LIN {X -0.244,Y -561.482,Z 954.741,A 0.000,B 0.000,C 90.000,E1 349.398} C_DIS
LIN {X 0.065,Y -565.954,Z 954.738,A 0.000,B 0.000,C 90.000,E1 348.814} C_DIS
LIN {X -0.209,Y -573.077,Z 954.733,A 0.000,B 0.000,C 90.000,E1 347.881} C_DIS
LIN {X -0.280,Y -579.380,Z 954.727,A 0.000,B 0.000,C 90.000,E1 346.937} C_DIS
LIN {X -0.174,Y -584.312,Z 954.723,A 0.000,B 0.000,C 90.000,E1 346.117} C_DIS
LIN {X -0.106,Y -589.678,Z 954.718,A 0.000,B 0.000,C 90.000,E1 345.172} C_DIS
LIN {X 0.183,Y -594.663,Z 954.712,A 0.000,B 0.000,C 90.000,E1 344.212} C_DIS
LIN {X 0.084,Y -600.569,Z 954.706,A 0.000,B 0.000,C 90.000,E1 343.032} C_DIS
LIN {X -0.062,Y -604.887,Z 954.701,A 0.000,B 0.000,C 90.000,E1 342.127} C_DIS
LIN {X 0.073,Y -608.439,Z 954.696,A 0.000,B 0.000,C 90.000,E1 341.329} C_DIS
LIN {X 0.049,Y -611.830,Z 954.692,A 0.000,B 0.000,C 90.000,E1 340.550} C_DIS
LIN {X 0.007,Y -616.058,Z 954.686,A 0.000,B 0.000,C 90.000,E1 339.518} C_DIS
LIN {X 0.265,Y -619.088,Z 954.682,A 0.000,B 0.000,C 90.000,E1 338.720} C_DIS
LIN {X -0.031,Y -622.893,Z 954.676,A 0.000,B 0.000,C 90.000,E1 337.720} C_DIS
LIN {X 0.305,Y -626.443,Z 954.671,A 0.000,B 0.000,C 90.000,E1 336.666} C_DIS
LIN {X 0.111,Y -629.800,Z 954.665,A 0.000,B 0.000,C 90.000,E1 335.665} C_DIS
LIN {X -0.044,Y -632.948,Z 954.659,A 0.000,B 0.000,C 90.000,E1 334.665} C_DIS
LIN {X 0.111,Y -635.819,Z 954.654,A 0.000,B 0.000,C 90.000,E1 333.640} C_DIS
LIN {X -0.205,Y -639.174,Z 954.647,A 0.000,B 0.000,C 90.000,E1 332.410} C_DIS
LIN {X 0.033,Y -641.563,Z 954.641,A 0.000,B 0.000,C 90.000,E1 331.385} C_DIS
LIN {X 0.118,Y -644.440,Z 954.634,A 0.000,B 0.000,C 90.000,E1 330.127} C_DIS
LIN {X 0.253,Y -646.929,Z 954.627,A 0.000,B 0.000,C 90.000,E1 328.869} C_DIS
LIN {X -0.207,Y -648.652,Z 954.622,A 0.000,B 0.000,C 90.000,E1 327.916} C_DIS
LIN {X 0.334,Y -650.629,Z 954.615,A 0.000,B 0.000,C 90.000,E1 326.628} C_DIS
LIN {X 0.361,Y -652.174,Z 954.608,A 0.000,B 0.000,C 90.000,E1 325.388} C_DIS
LIN {X 0.334,Y -653.400,Z 954.602,A 0.000,B 0.000,C 90.000,E1 324.402} C_DIS
LIN {X -0.139,Y -654.470,Z 954.596,A 0.000,B 0.000,C 90.000,E1 323.210} C_DIS
LIN {X 0.253,Y -655.293,Z 954.590,A 0.000,B 0.000,C 90.000,E1 322.190} C_DIS
LIN {X -0.315,Y -656.531,Z 954.581,A 0.000,B 0.000,C 90.000,E1 320.517} C_DIS
LIN {X 0.016,Y -657.478,Z 954.572,A 0.000,B 0.000,C 90.000,E1 319.013} C_DIS
LIN {X 0.167,Y -659.709,Z 954.555,A 0.000,B 0.000,C 90.000,E1 315.810} C_DIS
LIN {X 0.064,Y -660.674,Z 954.548,A 0.000,B 0.000,C 90.000,E1 314.595} C_DIS
LIN {X -0.063,Y -662.179,Z 954.538,A 0.000,B 0.000,C 90.000,E1 312.894} C_DIS
LIN {X 0.363,Y -663.736,Z 954.529,A 0.000,B 0.000,C 90.000,E1 311.148} C_DIS
LIN {X -0.090,Y -664.938,Z 954.521,A 0.000,B 0.000,C 90.000,E1 309.725} C_DIS
LIN {X -0.003,Y -666.013,Z 954.513,A 0.000,B 0.000,C 90.000,E1 308.257} C_DIS
LIN {X 0.022,Y -666.550,Z 954.507,A 0.000,B 0.000,C 90.000,E1 307.282} C_DIS
LIN {X -0.250,Y -667.011,Z 954.500,A 0.000,B 0.000,C 90.000,E1 306.091} C_DIS
LIN {X 0.424,Y -667.346,Z 954.494,A 0.000,B 0.000,C 90.000,E1 304.818} C_DIS
LIN {X -0.038,Y -668.158,Z 954.482,A 0.000,B 0.000,C 90.000,E1 302.673} C_DIS
LIN {X 0.293,Y -669.354,Z 954.469,A 0.000,B 0.000,C 90.000,E1 300.463} C_DIS
LIN {X 0.006,Y -671.420,Z 954.457,A 0.000,B 0.000,C 90.000,E1 298.309} C_DIS
LIN {X -0.153,Y -675.500,Z 954.443,A 0.000,B 0.000,C 90.000,E1 295.668} C_DIS
LIN {X -0.122,Y -677.621,Z 954.436,A 0.000,B 0.000,C 90.000,E1 294.463} C_DIS
LIN {X -0.065,Y -679.550,Z 954.429,A 0.000,B 0.000,C 90.000,E1 293.259} C_DIS
LIN {X 0.055,Y -680.122,Z 954.427,A 0.000,B 0.000,C 90.000,E1 292.770} C_DIS
LIN {X 0.182,Y -680.201,Z 954.424,A 0.000,B 0.000,C 90.000,E1 292.280} C_DIS
LIN {X -0.256,Y -680.187,Z 954.423,A 0.000,B 0.000,C 90.000,E1 292.078} C_DIS
LIN {X -0.319,Y -679.732,Z 954.421,A 0.000,B 0.000,C 90.000,E1 291.844} C_DIS
LIN {X -0.188,Y -678.464,Z 954.419,A 0.000,B 0.000,C 90.000,E1 291.354} C_DIS
LIN {X -0.096,Y -677.859,Z 954.418,A 0.000,B 0.000,C 90.000,E1 291.227} C_DIS
LIN {X 0.086,Y -675.944,Z 954.417,A 0.000,B 0.000,C 90.000,E1 290.972} C_DIS
LIN {X 0.150,Y -672.172,Z 954.415,A 0.000,B 0.000,C 90.000,E1 290.610} C_DIS
LIN {X 0.284,Y -670.597,Z 954.414,A 0.000,B 0.000,C 90.000,E1 290.482} C_DIS
LIN {X 0.022,Y -661.757,Z 954.411,A 0.000,B 0.000,C 90.000,E1 289.939} C_DIS
LIN {X -0.168,Y -659.824,Z 954.410,A 0.000,B 0.000,C 90.000,E1 289.812} C_DIS
LIN {X 0.108,Y -658.940,Z 954.409,A 0.000,B 0.000,C 90.000,E1 289.685} C_DIS
LIN {X 0.072,Y -658.929,Z 954.409,A 0.000,B 0.000,C 90.000,E1 289.685} C_DIS
LIN {X 0.021,Y -658.798,Z 954.409,A 0.000,B 0.000,C 90.000,E1 289.523} C_DIS
LIN {X 0.073,Y -659.029,Z 954.408,A 0.000,B 0.000,C 90.000,E1 289.396} C_DIS
LIN {X 0.012,Y -660.078,Z 954.406,A 0.000,B 0.000,C 90.000,E1 289.033} C_DIS
LIN {X 0.060,Y -663.109,Z 954.402,A 0.000,B 0.000,C 90.000,E1 288.417} C_DIS
LIN {X 0.174,Y -668.460,Z 954.397,A 0.000,B 0.000,C 90.000,E1 287.457} C_DIS
LIN {X 0.095,Y -669.821,Z 954.396,A 0.000,B 0.000,C 90.000,E1 287.221} C_DIS
LIN {X 0.074,Y -673.178,Z 954.392,A 0.000,B 0.000,C 90.000,E1 286.496} C_DIS
LIN {X -0.106,Y -675.937,Z 954.388,A 0.000,B 0.000,C 90.000,E1 285.788} C_DIS
LIN {X -0.029,Y -677.427,Z 954.385,A 0.000,B 0.000,C 90.000,E1 285.300} C_DIS
LIN {X -0.169,Y -679.177,Z 954.381,A 0.000,B 0.000,C 90.000,E1 284.592} C_DIS
LIN {X -0.289,Y -680.537,Z 954.377,A 0.000,B 0.000,C 90.000,E1 283.883} C_DIS
LIN {X 0.233,Y -682.070,Z 954.372,A 0.000,B 0.000,C 90.000,E1 282.883} C_DIS
LIN {X 0.168,Y -682.627,Z 954.369,A 0.000,B 0.000,C 90.000,E1 282.411} C_DIS
LIN {X -0.066,Y -683.123,Z 954.365,A 0.000,B 0.000,C 90.000,E1 281.715} C_DIS
LIN {X -0.125,Y -683.262,Z 954.362,A 0.000,B 0.000,C 90.000,E1 281.243} C_DIS
LIN {X -0.316,Y -683.055,Z 954.360,A 0.000,B 0.000,C 90.000,E1 280.782} C_DIS
LIN {X 0.293,Y -682.648,Z 954.357,A 0.000,B 0.000,C 90.000,E1 280.254} C_DIS
LIN {X 0.106,Y -681.924,Z 954.354,A 0.000,B 0.000,C 90.000,E1 279.792} C_DIS
LIN {X 0.068,Y -681.479,Z 954.353,A 0.000,B 0.000,C 90.000,E1 279.557} C_DIS
LIN {X -0.121,Y -680.255,Z 954.351,A 0.000,B 0.000,C 90.000,E1 279.095} C_DIS
LIN {X -0.213,Y -678.729,Z 954.348,A 0.000,B 0.000,C 90.000,E1 278.624} C_DIS
LIN {X 0.192,Y -675.923,Z 954.344,A 0.000,B 0.000,C 90.000,E1 277.871} C_DIS
LIN {X -0.110,Y -673.075,Z 954.341,A 0.000,B 0.000,C 90.000,E1 277.296} C_DIS
LIN {X 0.317,Y -670.504,Z 954.338,A 0.000,B 0.000,C 90.000,E1 276.777} C_DIS
LIN {X 0.059,Y -667.711,Z 954.335,A 0.000,B 0.000,C 90.000,E1 276.315} C_DIS
LIN {X -0.215,Y -664.623,Z 954.332,A 0.000,B 0.000,C 90.000,E1 275.853} C_DIS
LIN {X 0.058,Y -660.056,Z 954.329,A 0.000,B 0.000,C 90.000,E1 275.220} C_DIS
LIN {X 0.288,Y -654.936,Z 954.326,A 0.000,B 0.000,C 90.000,E1 274.588} C_DIS
LIN {X -0.014,Y -651.703,Z 954.324,A 0.000,B 0.000,C 90.000,E1 274.245} C_DIS
LIN {X 0.194,Y -645.675,Z 954.320,A 0.000,B 0.000,C 90.000,E1 273.612} C_DIS
LIN {X -0.125,Y -639.286,Z 954.317,A 0.000,B 0.000,C 90.000,E1 273.037} C_DIS
LIN {X -0.154,Y -632.639,Z 954.314,A 0.000,B 0.000,C 90.000,E1 272.465} C_DIS
LIN {X -0.117,Y -628.290,Z 954.312,A 0.000,B 0.000,C 90.000,E1 272.121} C_DIS
LIN {X 0.146,Y -623.990,Z 954.310,A 0.000,B 0.000,C 90.000,E1 271.776} C_DIS
LIN {X 0.090,Y -617.979,Z 954.308,A 0.000,B 0.000,C 90.000,E1 271.375} C_DIS
LIN {X -0.084,Y -610.095,Z 954.305,A 0.000,B 0.000,C 90.000,E1 270.917} C_DIS
LIN {X -0.267,Y -603.588,Z 954.303,A 0.000,B 0.000,C 90.000,E1 270.573} C_DIS
LIN {X -0.108,Y -596.754,Z 954.301,A 0.000,B 0.000,C 90.000,E1 270.229} C_DIS
LIN {X -0.054,Y -591.586,Z 954.300,A 0.000,B 0.000,C 90.000,E1 270.000} C_DIS
LIN {X 0.162,Y -584.378,Z 954.299,A 0.000,B 0.000,C 90.000,E1 269.714} C_DIS
LIN {X 0.133,Y -578.913,Z 954.298,A 0.000,B 0.000,C 90.000,E1 269.542} C_DIS
LIN {X -0.182,Y -571.139,Z 954.296,A 0.000,B 0.000,C 90.000,E1 269.370} C_DIS
LIN {X 0.260,Y -564.825,Z 954.296,A 0.000,B 0.000,C 90.000,E1 269.198} C_DIS
LIN {X -0.025,Y -557.881,Z 954.295,A 0.000,B 0.000,C 90.000,E1 269.141} C_DIS
LIN {X 0.065,Y -549.908,Z 954.295,A 0.000,B 0.000,C 90.000,E1 269.083} C_DIS
LIN {X -0.046,Y -548.727,Z 954.295,A 0.000,B 0.000,C 90.000,E1 269.083} C_DIS
LIN {X -0.084,Y -548.413,Z 954.295,A 0.000,B 0.000,C 90.000,E1 269.083} C_DIS
LIN {X -0.218,Y -543.489,Z 954.293,A 0.000,B 0.000,C 90.000,E1 268.740} C_DIS
LIN {X -0.251,Y -543.453,Z 954.293,A 0.000,B 0.000,C 90.000,E1 268.740} C_DIS
LIN {X -0.261,Y -542.935,Z 954.292,A 0.000,B 0.000,C 90.000,E1 268.511} C_DIS
LIN {X -0.023,Y -541.478,Z 954.282,A 0.000,B 0.000,C 90.000,E1 266.731} C_DIS
LIN {X 0.170,Y -540.033,Z 954.271,A 0.000,B 0.000,C 90.000,E1 264.723} C_DIS
LIN {X -0.177,Y -538.999,Z 954.263,A 0.000,B 0.000,C 90.000,E1 263.337} C_DIS
LIN {X -0.003,Y -538.008,Z 954.255,A 0.000,B 0.000,C 90.000,E1 261.894} C_DIS
LIN {X 0.164,Y -536.945,Z 954.249,A 0.000,B 0.000,C 90.000,E1 260.735} C_DIS
LIN {X -0.217,Y -535.611,Z 954.242,A 0.000,B 0.000,C 90.000,E1 259.634} C_DIS
LIN {X 0.199,Y -532.710,Z 954.230,A 0.000,B 0.000,C 90.000,E1 257.297} C_DIS
LIN {X 0.250,Y -529.932,Z 954.217,A 0.000,B 0.000,C 90.000,E1 254.991} C_DIS
LIN {X 0.177,Y -527.986,Z 954.207,A 0.000,B 0.000,C 90.000,E1 253.268} C_DIS
LIN {X 0.204,Y -526.299,Z 954.199,A 0.000,B 0.000,C 90.000,E1 251.819} C_DIS
LIN {X 0.204,Y -524.517,Z 954.191,A 0.000,B 0.000,C 90.000,E1 250.369} C_DIS
LIN {X -0.144,Y -522.628,Z 954.183,A 0.000,B 0.000,C 90.000,E1 248.954} C_DIS
LIN {X 0.112,Y -520.335,Z 954.173,A 0.000,B 0.000,C 90.000,E1 247.177} C_DIS
LIN {X -0.256,Y -518.649,Z 954.167,A 0.000,B 0.000,C 90.000,E1 246.049} C_DIS
LIN {X -0.165,Y -515.883,Z 954.157,A 0.000,B 0.000,C 90.000,E1 244.280} C_DIS
LIN {X -0.022,Y -513.574,Z 954.149,A 0.000,B 0.000,C 90.000,E1 242.794} C_DIS
LIN {X -0.274,Y -510.727,Z 954.139,A 0.000,B 0.000,C 90.000,E1 241.051} C_DIS
LIN {X 0.045,Y -509.196,Z 954.134,A 0.000,B 0.000,C 90.000,E1 240.127} C_DIS
LIN {X 0.187,Y -505.896,Z 954.124,A 0.000,B 0.000,C 90.000,E1 238.329} C_DIS
LIN {X 0.208,Y -502.650,Z 954.116,A 0.000,B 0.000,C 90.000,E1 236.834} C_DIS
LIN {X -0.129,Y -499.952,Z 954.109,A 0.000,B 0.000,C 90.000,E1 235.674} C_DIS
LIN {X -0.085,Y -495.819,Z 954.099,A 0.000,B 0.000,C 90.000,E1 233.863} C_DIS
LIN {X 0.050,Y -493.152,Z 954.093,A 0.000,B 0.000,C 90.000,E1 232.637} C_DIS
LIN {X -0.013,Y -489.753,Z 954.084,A 0.000,B 0.000,C 90.000,E1 231.126} C_DIS
LIN {X -0.212,Y -486.249,Z 954.076,A 0.000,B 0.000,C 90.000,E1 229.622} C_DIS
LIN {X -0.212,Y -481.290,Z 954.064,A 0.000,B 0.000,C 90.000,E1 227.472} C_DIS
LIN {X -0.159,Y -479.200,Z 954.058,A 0.000,B 0.000,C 90.000,E1 226.539} C_DIS
LIN {X -0.249,Y -475.792,Z 954.050,A 0.000,B 0.000,C 90.000,E1 225.000} C_DIS
LIN {X 0.127,Y -470.977,Z 954.038,A 0.000,B 0.000,C 90.000,E1 222.771} C_DIS
LIN {X -0.028,Y -466.887,Z 954.027,A 0.000,B 0.000,C 90.000,E1 220.906} C_DIS
LIN {X 0.167,Y -461.987,Z 954.015,A 0.000,B 0.000,C 90.000,E1 218.669} C_DIS
LIN {X 0.183,Y -458.509,Z 954.006,A 0.000,B 0.000,C 90.000,E1 217.076} C_DIS
LIN {X -0.042,Y -454.181,Z 953.995,A 0.000,B 0.000,C 90.000,E1 215.185} C_DIS
LIN {X 0.015,Y -449.974,Z 953.985,A 0.000,B 0.000,C 90.000,E1 213.245} C_DIS
LIN {X -0.274,Y -445.728,Z 953.974,A 0.000,B 0.000,C 90.000,E1 211.337} C_DIS
LIN {X -0.018,Y -442.885,Z 953.967,A 0.000,B 0.000,C 90.000,E1 210.001} C_DIS
LIN {X -0.117,Y -437.955,Z 953.954,A 0.000,B 0.000,C 90.000,E1 207.719} C_DIS
LIN {X 0.004,Y -434.323,Z 953.945,A 0.000,B 0.000,C 90.000,E1 206.052} C_DIS
LIN {X 0.046,Y -430.643,Z 953.936,A 0.000,B 0.000,C 90.000,E1 204.387} C_DIS
LIN {X 0.017,Y -426.073,Z 953.924,A 0.000,B 0.000,C 90.000,E1 202.386} C_DIS
LIN {X 0.096,Y -419.500,Z 953.908,A 0.000,B 0.000,C 90.000,E1 199.341} C_DIS
LIN {X 0.065,Y -413.978,Z 953.892,A 0.000,B 0.000,C 90.000,E1 196.622} C_DIS
LIN {X 0.135,Y -410.602,Z 953.883,A 0.000,B 0.000,C 90.000,E1 194.898} C_DIS
LIN {X 0.143,Y -406.413,Z 953.871,A 0.000,B 0.000,C 90.000,E1 192.827} C_DIS
LIN {X -0.131,Y -403.062,Z 953.862,A 0.000,B 0.000,C 90.000,E1 191.130} C_DIS
LIN {X -0.067,Y -400.456,Z 953.854,A 0.000,B 0.000,C 90.000,E1 189.726} C_DIS
LIN {X -0.200,Y -397.084,Z 953.844,A 0.000,B 0.000,C 90.000,E1 187.992} C_DIS
LIN {X -0.041,Y -393.117,Z 953.833,A 0.000,B 0.000,C 90.000,E1 185.853} C_DIS
LIN {X -0.021,Y -387.360,Z 953.813,A 0.000,B 0.000,C 90.000,E1 182.293} C_DIS
LIN {X 0.089,Y -386.414,Z 953.807,A 0.000,B 0.000,C 90.000,E1 181.203} C_DIS
LIN {X -0.109,Y -386.020,Z 953.803,A 0.000,B 0.000,C 90.000,E1 180.516} C_DIS
LIN {X 0.177,Y -385.993,Z 953.801,A 0.000,B 0.000,C 90.000,E1 180.115} C_DIS
LIN {X 0.076,Y -386.144,Z 953.799,A 0.000,B 0.000,C 90.000,E1 179.771} C_DIS
LIN {X -0.126,Y -387.039,Z 953.795,A 0.000,B 0.000,C 90.000,E1 179.083} C_DIS
LIN {X 0.071,Y -388.893,Z 953.791,A 0.000,B 0.000,C 90.000,E1 178.339} C_DIS
LIN {X 0.083,Y -390.263,Z 953.789,A 0.000,B 0.000,C 90.000,E1 177.993} C_DIS
LIN {X -0.008,Y -392.230,Z 953.787,A 0.000,B 0.000,C 90.000,E1 177.650} C_DIS
LIN {X -0.092,Y -394.356,Z 953.785,A 0.000,B 0.000,C 90.000,E1 177.306} C_DIS
LIN {X -0.170,Y -397.323,Z 953.783,A 0.000,B 0.000,C 90.000,E1 176.963} C_DIS
LIN {X -0.101,Y -399.882,Z 953.781,A 0.000,B 0.000,C 90.000,E1 176.674} C_DIS
LIN {X -0.205,Y -407.252,Z 953.778,A 0.000,B 0.000,C 90.000,E1 175.988} C_DIS
LIN {X -0.189,Y -413.386,Z 953.775,A 0.000,B 0.000,C 90.000,E1 175.469} C_DIS
LIN {X 0.047,Y -430.440,Z 953.767,A 0.000,B 0.000,C 90.000,E1 173.970} C_DIS
LIN {X -0.025,Y -440.720,Z 953.761,A 0.000,B 0.000,C 90.000,E1 173.053} C_DIS
LIN {X -0.183,Y -449.544,Z 953.757,A 0.000,B 0.000,C 90.000,E1 172.243} C_DIS
LIN {X -0.029,Y -455.300,Z 953.754,A 0.000,B 0.000,C 90.000,E1 171.659} C_DIS
LIN {X -0.017,Y -461.063,Z 953.750,A 0.000,B 0.000,C 90.000,E1 171.084} C_DIS
LIN {X 0.171,Y -470.266,Z 953.745,A 0.000,B 0.000,C 90.000,E1 170.095} C_DIS
LIN {X -0.112,Y -478.133,Z 953.740,A 0.000,B 0.000,C 90.000,E1 169.218} C_DIS
LIN {X 0.139,Y -483.329,Z 953.737,A 0.000,B 0.000,C 90.000,E1 168.578} C_DIS
LIN {X 0.000,Y -489.497,Z 953.732,A 0.000,B 0.000,C 90.000,E1 167.825} C_DIS
LIN {X 0.170,Y -493.049,Z 953.730,A 0.000,B 0.000,C 90.000,E1 167.353} C_DIS
LIN {X -0.085,Y -502.168,Z 953.723,A 0.000,B 0.000,C 90.000,E1 166.172} C_DIS
LIN {X 0.127,Y -509.493,Z 953.717,A 0.000,B 0.000,C 90.000,E1 165.102} C_DIS
LIN {X -0.031,Y -518.221,Z 953.710,A 0.000,B 0.000,C 90.000,E1 163.795} C_DIS
LIN {X -0.104,Y -524.764,Z 953.704,A 0.000,B 0.000,C 90.000,E1 162.779} C_DIS
LIN {X 0.082,Y -532.828,Z 953.697,A 0.000,B 0.000,C 90.000,E1 161.456} C_DIS
LIN {X 0.036,Y -539.926,Z 953.691,A 0.000,B 0.000,C 90.000,E1 160.315} C_DIS
LIN {X 0.218,Y -545.003,Z 953.686,A 0.000,B 0.000,C 90.000,E1 159.444} C_DIS
LIN {X -0.096,Y -552.593,Z 953.679,A 0.000,B 0.000,C 90.000,E1 158.209} C_DIS
LIN {X 0.216,Y -559.724,Z 953.672,A 0.000,B 0.000,C 90.000,E1 156.922} C_DIS
LIN {X 0.218,Y -563.457,Z 953.668,A 0.000,B 0.000,C 90.000,E1 156.230} C_DIS
LIN {X -0.018,Y -569.148,Z 953.662,A 0.000,B 0.000,C 90.000,E1 155.153} C_DIS
LIN {X -0.015,Y -573.176,Z 953.657,A 0.000,B 0.000,C 90.000,E1 154.332} C_DIS
LIN {X -0.270,Y -579.305,Z 953.650,A 0.000,B 0.000,C 90.000,E1 152.999} C_DIS
LIN {X 0.161,Y -582.199,Z 953.646,A 0.000,B 0.000,C 90.000,E1 152.281} C_DIS
LIN {X -0.081,Y -586.471,Z 953.640,A 0.000,B 0.000,C 90.000,E1 151.229} C_DIS
LIN {X 0.251,Y -590.483,Z 953.634,A 0.000,B 0.000,C 90.000,E1 150.127} C_DIS
LIN {X 0.014,Y -595.289,Z 953.627,A 0.000,B 0.000,C 90.000,E1 148.820} C_DIS
LIN {X -0.260,Y -598.936,Z 953.621,A 0.000,B 0.000,C 90.000,E1 147.788} C_DIS
LIN {X -0.061,Y -605.071,Z 953.611,A 0.000,B 0.000,C 90.000,E1 145.928} C_DIS
LIN {X -0.193,Y -608.604,Z 953.605,A 0.000,B 0.000,C 90.000,E1 144.895} C_DIS
LIN {X -0.203,Y -613.893,Z 953.596,A 0.000,B 0.000,C 90.000,E1 143.336} C_DIS
LIN {X -0.289,Y -619.907,Z 953.586,A 0.000,B 0.000,C 90.000,E1 141.537} C_DIS
LIN {X -0.037,Y -624.171,Z 953.579,A 0.000,B 0.000,C 90.000,E1 140.231} C_DIS
LIN {X -0.048,Y -630.122,Z 953.569,A 0.000,B 0.000,C 90.000,E1 138.447} C_DIS
LIN {X 0.103,Y -636.518,Z 953.559,A 0.000,B 0.000,C 90.000,E1 136.662} C_DIS
LIN {X 0.100,Y -641.015,Z 953.552,A 0.000,B 0.000,C 90.000,E1 135.405} C_DIS
LIN {X -0.365,Y -646.462,Z 953.544,A 0.000,B 0.000,C 90.000,E1 133.947} C_DIS
LIN {X -0.264,Y -651.876,Z 953.536,A 0.000,B 0.000,C 90.000,E1 132.447} C_DIS
LIN {X -0.040,Y -658.342,Z 953.526,A 0.000,B 0.000,C 90.000,E1 130.701} C_DIS
LIN {X -0.128,Y -662.979,Z 953.519,A 0.000,B 0.000,C 90.000,E1 129.483} C_DIS
LIN {X -0.047,Y -667.602,Z 953.513,A 0.000,B 0.000,C 90.000,E1 128.257} C_DIS
LIN {X 0.003,Y -671.201,Z 953.507,A 0.000,B 0.000,C 90.000,E1 127.282} C_DIS
LIN {X 0.225,Y -674.629,Z 953.502,A 0.000,B 0.000,C 90.000,E1 126.297} C_DIS
LIN {X -0.054,Y -677.888,Z 953.496,A 0.000,B 0.000,C 90.000,E1 125.358} C_DIS
LIN {X 0.426,Y -681.673,Z 953.490,A 0.000,B 0.000,C 90.000,E1 124.119} C_DIS
LIN {X 0.029,Y -685.100,Z 953.483,A 0.000,B 0.000,C 90.000,E1 122.959} C_DIS
LIN {X 0.054,Y -687.590,Z 953.478,A 0.000,B 0.000,C 90.000,E1 122.005} C_DIS
LIN {X 0.108,Y -689.928,Z 953.473,A 0.000,B 0.000,C 90.000,E1 121.052} C_DIS
LIN {X 0.197,Y -691.468,Z 953.469,A 0.000,B 0.000,C 90.000,E1 120.335} C_DIS
LIN {X 0.069,Y -692.442,Z 953.466,A 0.000,B 0.000,C 90.000,E1 119.873} C_DIS
LIN {X -0.171,Y -694.023,Z 953.461,A 0.000,B 0.000,C 90.000,E1 118.949} C_DIS
LIN {X -0.036,Y -695.058,Z 953.457,A 0.000,B 0.000,C 90.000,E1 118.231} C_DIS
LIN {X 0.363,Y -696.072,Z 953.452,A 0.000,B 0.000,C 90.000,E1 117.257} C_DIS
LIN {X 0.096,Y -696.838,Z 953.445,A 0.000,B 0.000,C 90.000,E1 116.104} C_DIS
LIN {X -0.165,Y -697.205,Z 953.439,A 0.000,B 0.000,C 90.000,E1 114.951} C_DIS
LIN {X 0.321,Y -697.234,Z 953.435,A 0.000,B 0.000,C 90.000,E1 114.207} C_DIS
LIN {X -0.081,Y -696.974,Z 953.432,A 0.000,B 0.000,C 90.000,E1 113.770} C_DIS
LIN {X 0.156,Y -695.919,Z 953.429,A 0.000,B 0.000,C 90.000,E1 113.281} C_DIS
LIN {X -0.230,Y -695.143,Z 953.428,A 0.000,B 0.000,C 90.000,E1 113.078} C_DIS
LIN {X -0.004,Y -692.316,Z 953.426,A 0.000,B 0.000,C 90.000,E1 112.589} C_DIS
LIN {X 0.116,Y -691.505,Z 953.425,A 0.000,B 0.000,C 90.000,E1 112.461} C_DIS
LIN {X 0.235,Y -690.348,Z 953.424,A 0.000,B 0.000,C 90.000,E1 112.333} C_DIS
LIN {X 0.349,Y -688.559,Z 953.424,A 0.000,B 0.000,C 90.000,E1 112.206} C_DIS
LIN {X -0.193,Y -683.327,Z 953.422,A 0.000,B 0.000,C 90.000,E1 111.972} C_DIS
LIN {X -0.287,Y -681.532,Z 953.422,A 0.000,B 0.000,C 90.000,E1 111.897} C_DIS
LIN {X 0.198,Y -677.217,Z 953.421,A 0.000,B 0.000,C 90.000,E1 111.716} C_DIS
LIN {X 0.148,Y -674.161,Z 953.420,A 0.000,B 0.000,C 90.000,E1 111.663} C_DIS
LIN {X 0.387,Y -667.380,Z 953.420,A 0.000,B 0.000,C 90.000,E1 111.589} C_DIS
LIN {X 0.319,Y -632.121,Z 953.420,A 0.000,B 0.000,C 90.000,E1 111.589} C_DIS
LIN {X -0.262,Y -627.805,Z 953.420,A 0.000,B 0.000,C 90.000,E1 111.589} C_DIS
LIN {X 0.027,Y -622.129,Z 953.419,A 0.000,B 0.000,C 90.000,E1 111.461} C_DIS
LIN {X -0.010,Y -615.215,Z 953.418,A 0.000,B 0.000,C 90.000,E1 111.280} C_DIS
LIN {X 0.194,Y -607.245,Z 953.417,A 0.000,B 0.000,C 90.000,E1 110.972} C_DIS
LIN {X -0.121,Y -599.399,Z 953.414,A 0.000,B 0.000,C 90.000,E1 110.610} C_DIS
LIN {X -0.139,Y -594.282,Z 953.413,A 0.000,B 0.000,C 90.000,E1 110.301} C_DIS
LIN {X -0.056,Y -577.074,Z 953.406,A 0.000,B 0.000,C 90.000,E1 109.033} C_DIS
LIN {X 0.286,Y -573.355,Z 953.405,A 0.000,B 0.000,C 90.000,E1 108.779} C_DIS
LIN {X -0.057,Y -568.575,Z 953.403,A 0.000,B 0.000,C 90.000,E1 108.544} C_DIS
LIN {X -0.099,Y -556.788,Z 953.400,A 0.000,B 0.000,C 90.000,E1 108.000} C_DIS
LIN {X -0.205,Y -553.162,Z 953.399,A 0.000,B 0.000,C 90.000,E1 107.819} C_DIS
LIN {X 0.017,Y -551.533,Z 953.398,A 0.000,B 0.000,C 90.000,E1 107.638} C_DIS
LIN {X -0.023,Y -551.496,Z 953.398,A 0.000,B 0.000,C 90.000,E1 107.638} C_DIS
LIN {X 0.100,Y -551.025,Z 953.397,A 0.000,B 0.000,C 90.000,E1 107.402} C_DIS
LIN {X -0.062,Y -550.901,Z 953.394,A 0.000,B 0.000,C 90.000,E1 106.858} C_DIS
LIN {X -0.186,Y -551.549,Z 953.384,A 0.000,B 0.000,C 90.000,E1 105.190} C_DIS
LIN {X 0.043,Y -552.821,Z 953.370,A 0.000,B 0.000,C 90.000,E1 102.647} C_DIS
LIN {X -0.063,Y -554.573,Z 953.358,A 0.000,B 0.000,C 90.000,E1 100.423} C_DIS
LIN {X -0.199,Y -555.592,Z 953.352,A 0.000,B 0.000,C 90.000,E1 99.321} C_DIS
LIN {X -0.135,Y -557.097,Z 953.342,A 0.000,B 0.000,C 90.000,E1 97.644} C_DIS
LIN {X -0.171,Y -558.239,Z 953.335,A 0.000,B 0.000,C 90.000,E1 96.258} C_DIS
LIN {X -0.245,Y -559.174,Z 953.327,A 0.000,B 0.000,C 90.000,E1 94.878} C_DIS
LIN {X -0.214,Y -560.159,Z 953.318,A 0.000,B 0.000,C 90.000,E1 93.212} C_DIS
LIN {X -0.267,Y -560.902,Z 953.310,A 0.000,B 0.000,C 90.000,E1 91.833} C_DIS
LIN {X 0.212,Y -561.512,Z 953.302,A 0.000,B 0.000,C 90.000,E1 90.401} C_DIS
LIN {X 0.045,Y -561.880,Z 953.296,A 0.000,B 0.000,C 90.000,E1 89.312} C_DIS
LIN {X 0.097,Y -562.239,Z 953.287,A 0.000,B 0.000,C 90.000,E1 87.650} C_DIS
LIN {X -0.043,Y -562.489,Z 953.281,A 0.000,B 0.000,C 90.000,E1 86.560} C_DIS
LIN {X -0.042,Y -562.749,Z 953.273,A 0.000,B 0.000,C 90.000,E1 85.179} C_DIS
LIN {X 0.198,Y -563.015,Z 953.263,A 0.000,B 0.000,C 90.000,E1 83.223} C_DIS
LIN {X 0.093,Y -563.492,Z 953.250,A 0.000,B 0.000,C 90.000,E1 81.027} C_DIS
LIN {X -0.210,Y -564.441,Z 953.236,A 0.000,B 0.000,C 90.000,E1 78.578} C_DIS
LIN {X 0.018,Y -565.644,Z 953.224,A 0.000,B 0.000,C 90.000,E1 76.353} C_DIS
LIN {X 0.059,Y -566.723,Z 953.215,A 0.000,B 0.000,C 90.000,E1 74.700} C_DIS
LIN {X 0.054,Y -567.983,Z 953.204,A 0.000,B 0.000,C 90.000,E1 72.779} C_DIS
LIN {X -0.034,Y -568.643,Z 953.198,A 0.000,B 0.000,C 90.000,E1 71.692} C_DIS
LIN {X -0.112,Y -569.260,Z 953.192,A 0.000,B 0.000,C 90.000,E1 70.604} C_DIS
LIN {X 0.158,Y -569.821,Z 953.185,A 0.000,B 0.000,C 90.000,E1 69.209} C_DIS
LIN {X 0.108,Y -570.285,Z 953.177,A 0.000,B 0.000,C 90.000,E1 67.847} C_DIS
LIN {X 0.066,Y -570.668,Z 953.169,A 0.000,B 0.000,C 90.000,E1 66.485} C_DIS
LIN {X 0.087,Y -571.066,Z 953.160,A 0.000,B 0.000,C 90.000,E1 64.845} C_DIS
LIN {X 0.110,Y -571.353,Z 953.151,A 0.000,B 0.000,C 90.000,E1 63.204} C_DIS
LIN {X 0.044,Y -571.509,Z 953.144,A 0.000,B 0.000,C 90.000,E1 61.847} C_DIS
LIN {X 0.086,Y -571.556,Z 953.135,A 0.000,B 0.000,C 90.000,E1 60.205} C_DIS
LIN {X -0.243,Y -571.763,Z 953.124,A 0.000,B 0.000,C 90.000,E1 58.329} C_DIS
LIN {X 0.268,Y -571.663,Z 953.116,A 0.000,B 0.000,C 90.000,E1 56.914} C_DIS
LIN {X -0.182,Y -571.297,Z 953.109,A 0.000,B 0.000,C 90.000,E1 55.595} C_DIS
LIN {X 0.025,Y -570.944,Z 953.103,A 0.000,B 0.000,C 90.000,E1 54.482} C_DIS
LIN {X 0.292,Y -570.754,Z 953.100,A 0.000,B 0.000,C 90.000,E1 53.909} C_DIS
LIN {X -0.107,Y -570.321,Z 953.095,A 0.000,B 0.000,C 90.000,E1 53.130} C_DIS
LIN {X -0.033,Y -569.457,Z 953.089,A 0.000,B 0.000,C 90.000,E1 52.029} C_DIS
LIN {X 0.033,Y -568.445,Z 953.083,A 0.000,B 0.000,C 90.000,E1 50.928} C_DIS
LIN {X 0.082,Y -567.233,Z 953.077,A 0.000,B 0.000,C 90.000,E1 49.828} C_DIS
LIN {X -0.007,Y -566.176,Z 953.072,A 0.000,B 0.000,C 90.000,E1 49.013} C_DIS
LIN {X 0.263,Y -564.866,Z 953.068,A 0.000,B 0.000,C 90.000,E1 48.162} C_DIS
LIN {X 0.199,Y -562.811,Z 953.062,A 0.000,B 0.000,C 90.000,E1 47.067} C_DIS
LIN {X -0.036,Y -561.678,Z 953.059,A 0.000,B 0.000,C 90.000,E1 46.539} C_DIS
LIN {X 0.106,Y -560.484,Z 953.056,A 0.000,B 0.000,C 90.000,E1 45.972} C_DIS
LIN {X -0.090,Y -558.380,Z 953.051,A 0.000,B 0.000,C 90.000,E1 45.162} C_DIS
LIN {X 0.031,Y -556.855,Z 953.048,A 0.000,B 0.000,C 90.000,E1 44.595} C_DIS
LIN {X -0.202,Y -554.269,Z 953.043,A 0.000,B 0.000,C 90.000,E1 43.785} C_DIS
LIN {X -0.114,Y -552.448,Z 953.040,A 0.000,B 0.000,C 90.000,E1 43.218} C_DIS
LIN {X 0.005,Y -549.347,Z 953.035,A 0.000,B 0.000,C 90.000,E1 42.366} C_DIS
LIN {X -0.314,Y -547.132,Z 953.032,A 0.000,B 0.000,C 90.000,E1 41.838} C_DIS
LIN {X 0.320,Y -543.960,Z 953.028,A 0.000,B 0.000,C 90.000,E1 41.067} C_DIS
LIN {X 0.150,Y -540.627,Z 953.024,A 0.000,B 0.000,C 90.000,E1 40.378} C_DIS
LIN {X 0.185,Y -537.684,Z 953.021,A 0.000,B 0.000,C 90.000,E1 39.806} C_DIS
LIN {X -0.211,Y -534.592,Z 953.018,A 0.000,B 0.000,C 90.000,E1 39.277} C_DIS
LIN {X 0.120,Y -531.363,Z 953.015,A 0.000,B 0.000,C 90.000,E1 38.669} C_DIS
LIN {X 0.044,Y -524.446,Z 953.009,A 0.000,B 0.000,C 90.000,E1 37.523} C_DIS
LIN {X 0.104,Y -519.869,Z 953.005,A 0.000,B 0.000,C 90.000,E1 36.790} C_DIS
LIN {X -0.003,Y -516.046,Z 953.001,A 0.000,B 0.000,C 90.000,E1 36.217} C_DIS
LIN {X 0.200,Y -510.042,Z 952.996,A 0.000,B 0.000,C 90.000,E1 35.311} C_DIS
LIN {X -0.081,Y -503.432,Z 952.991,A 0.000,B 0.000,C 90.000,E1 34.452} C_DIS
LIN {X 0.103,Y -498.578,Z 952.988,A 0.000,B 0.000,C 90.000,E1 33.833} C_DIS
LIN {X 0.043,Y -492.112,Z 952.984,A 0.000,B 0.000,C 90.000,E1 33.086} C_DIS
LIN {X 0.146,Y -488.060,Z 952.981,A 0.000,B 0.000,C 90.000,E1 32.625} C_DIS
LIN {X 0.045,Y -481.018,Z 952.977,A 0.000,B 0.000,C 90.000,E1 31.926} C_DIS
LIN {X -0.186,Y -473.908,Z 952.974,A 0.000,B 0.000,C 90.000,E1 31.258} C_DIS
LIN {X 0.243,Y -463.529,Z 952.968,A 0.000,B 0.000,C 90.000,E1 30.256} C_DIS
LIN {X -0.015,Y -456.022,Z 952.965,A 0.000,B 0.000,C 90.000,E1 29.617} C_DIS
LIN {X -0.212,Y -443.997,Z 952.959,A 0.000,B 0.000,C 90.000,E1 28.615} C_DIS
LIN {X 0.107,Y -424.255,Z 952.949,A 0.000,B 0.000,C 90.000,E1 26.873} C_DIS
LIN {X -0.033,Y -407.876,Z 952.941,A 0.000,B 0.000,C 90.000,E1 25.335} C_DIS
LIN {X -0.079,Y -400.514,Z 952.937,A 0.000,B 0.000,C 90.000,E1 24.591} C_DIS
LIN {X -0.012,Y -395.559,Z 952.933,A 0.000,B 0.000,C 90.000,E1 24.003} C_DIS
LIN {X -0.240,Y -393.765,Z 952.932,A 0.000,B 0.000,C 90.000,E1 23.770} C_DIS
LIN {X -0.085,Y -392.059,Z 952.930,A 0.000,B 0.000,C 90.000,E1 23.462} C_DIS
LIN {X 0.014,Y -390.747,Z 952.929,A 0.000,B 0.000,C 90.000,E1 23.131} C_DIS
LIN {X -0.038,Y -390.132,Z 952.927,A 0.000,B 0.000,C 90.000,E1 22.898} C_DIS
LIN {X 0.147,Y -389.392,Z 952.924,A 0.000,B 0.000,C 90.000,E1 22.280} C_DIS
LIN {X 0.037,Y -389.598,Z 952.918,A 0.000,B 0.000,C 90.000,E1 21.227} C_DIS
LIN {X 0.012,Y -394.764,Z 952.888,A 0.000,B 0.000,C 90.000,E1 15.898} C_DIS
LIN {X 0.097,Y -398.370,Z 952.873,A 0.000,B 0.000,C 90.000,E1 13.063} C_DIS
LIN {X 0.125,Y -403.129,Z 952.855,A 0.000,B 0.000,C 90.000,E1 9.905} C_DIS
LIN {X 0.143,Y -406.696,Z 952.844,A 0.000,B 0.000,C 90.000,E1 7.814} C_DIS
LIN {X 0.142,Y -411.909,Z 952.828,A 0.000,B 0.000,C 90.000,E1 5.049} C_DIS
LIN {X -0.164,Y -417.693,Z 952.813,A 0.000,B 0.000,C 90.000,E1 2.350} C_DIS
LIN {X 0.207,Y -424.660,Z 952.797,A 0.000,B 0.000,C 90.000,E1 359.427} C_DIS
LIN {X -0.168,Y -425.684,Z 952.795,A 0.000,B 0.000,C 90.000,E1 359.141} C_DIS
LIN {X -0.105,Y -428.198,Z 952.792,A 0.000,B 0.000,C 90.000,E1 358.568} C_DIS
LIN {X -0.043,Y -430.272,Z 952.790,A 0.000,B 0.000,C 90.000,E1 358.224} C_DIS
LIN {X 0.046,Y -434.368,Z 952.788,A 0.000,B 0.000,C 90.000,E1 357.764} C_DIS
LIN {X 0.051,Y -435.779,Z 952.787,A 0.000,B 0.000,C 90.000,E1 357.650} C_DIS
LIN {X 0.163,Y -440.898,Z 952.785,A 0.000,B 0.000,C 90.000,E1 357.306} C_DIS
LIN {X -0.065,Y -453.945,Z 952.782,A 0.000,B 0.000,C 90.000,E1 356.674} C_DIS
LIN {X -0.028,Y -466.967,Z 952.778,A 0.000,B 0.000,C 90.000,E1 355.988} C_DIS
LIN {X -0.125,Y -480.098,Z 952.774,A 0.000,B 0.000,C 90.000,E1 355.298} C_DIS
LIN {X 0.221,Y -493.049,Z 952.770,A 0.000,B 0.000,C 90.000,E1 354.552} C_DIS
LIN {X 0.224,Y -501.257,Z 952.767,A 0.000,B 0.000,C 90.000,E1 354.090} C_DIS
LIN {X 0.228,Y -510.957,Z 952.764,A 0.000,B 0.000,C 90.000,E1 353.514} C_DIS
LIN {X 0.055,Y -518.522,Z 952.761,A 0.000,B 0.000,C 90.000,E1 353.053} C_DIS
LIN {X 0.234,Y -527.600,Z 952.758,A 0.000,B 0.000,C 90.000,E1 352.413} C_DIS
LIN {X -0.093,Y -536.355,Z 952.754,A 0.000,B 0.000,C 90.000,E1 351.781} C_DIS
LIN {X -0.131,Y -542.080,Z 952.752,A 0.000,B 0.000,C 90.000,E1 351.310} C_DIS
LIN {X -0.274,Y -548.611,Z 952.748,A 0.000,B 0.000,C 90.000,E1 350.735} C_DIS
LIN {X 0.059,Y -555.043,Z 952.745,A 0.000,B 0.000,C 90.000,E1 350.038} C_DIS
LIN {X 0.139,Y -561.125,Z 952.741,A 0.000,B 0.000,C 90.000,E1 349.342} C_DIS
LIN {X -0.107,Y -565.628,Z 952.738,A 0.000,B 0.000,C 90.000,E1 348.814} C_DIS
LIN {X -0.014,Y -570.805,Z 952.734,A 0.000,B 0.000,C 90.000,E1 348.117} C_DIS
LIN {X -0.196,Y -574.694,Z 952.731,A 0.000,B 0.000,C 90.000,E1 347.589} C_DIS
LIN {X -0.007,Y -580.078,Z 952.726,A 0.000,B 0.000,C 90.000,E1 346.756} C_DIS
LIN {X 0.017,Y -585.700,Z 952.721,A 0.000,B 0.000,C 90.000,E1 345.811} C_DIS
LIN {X 0.190,Y -590.326,Z 952.717,A 0.000,B 0.000,C 90.000,E1 344.991} C_DIS
LIN {X -0.010,Y -594.560,Z 952.712,A 0.000,B 0.000,C 90.000,E1 344.212} C_DIS
LIN {X 0.120,Y -599.864,Z 952.706,A 0.000,B 0.000,C 90.000,E1 343.142} C_DIS
LIN {X -0.030,Y -604.256,Z 952.701,A 0.000,B 0.000,C 90.000,E1 342.236} C_DIS
LIN {X -0.087,Y -607.855,Z 952.697,A 0.000,B 0.000,C 90.000,E1 341.456} C_DIS
LIN {X -0.119,Y -611.319,Z 952.693,A 0.000,B 0.000,C 90.000,E1 340.678} C_DIS
LIN {X 0.041,Y -615.558,Z 952.687,A 0.000,B 0.000,C 90.000,E1 339.625} C_DIS
LIN {X 0.076,Y -618.672,Z 952.683,A 0.000,B 0.000,C 90.000,E1 338.847} C_DIS
LIN {X -0.229,Y -622.496,Z 952.677,A 0.000,B 0.000,C 90.000,E1 337.847} C_DIS
LIN {X 0.098,Y -626.140,Z 952.671,A 0.000,B 0.000,C 90.000,E1 336.794} C_DIS
LIN {X -0.102,Y -629.561,Z 952.666,A 0.000,B 0.000,C 90.000,E1 335.793} C_DIS
LIN {X -0.229,Y -633.483,Z 952.658,A 0.000,B 0.000,C 90.000,E1 334.537} C_DIS
LIN {X -0.067,Y -636.347,Z 952.653,A 0.000,B 0.000,C 90.000,E1 333.512} C_DIS
LIN {X 0.193,Y -639.694,Z 952.646,A 0.000,B 0.000,C 90.000,E1 332.231} C_DIS
LIN {X -0.131,Y -642.076,Z 952.640,A 0.000,B 0.000,C 90.000,E1 331.257} C_DIS
LIN {X -0.039,Y -644.945,Z 952.633,A 0.000,B 0.000,C 90.000,E1 329.999} C_DIS
LIN {X 0.026,Y -646.958,Z 952.628,A 0.000,B 0.000,C 90.000,E1 328.997} C_DIS
LIN {X 0.118,Y -648.705,Z 952.622,A 0.000,B 0.000,C 90.000,E1 327.995} C_DIS
LIN {X -0.320,Y -650.331,Z 952.617,A 0.000,B 0.000,C 90.000,E1 327.041} C_DIS
LIN {X -0.276,Y -651.401,Z 952.613,A 0.000,B 0.000,C 90.000,E1 326.294} C_DIS
LIN {X -0.256,Y -653.574,Z 952.603,A 0.000,B 0.000,C 90.000,E1 324.562} C_DIS
LIN {X 0.117,Y -654.489,Z 952.598,A 0.000,B 0.000,C 90.000,E1 323.543} C_DIS
LIN {X 0.116,Y -655.707,Z 952.589,A 0.000,B 0.000,C 90.000,E1 322.065} C_DIS
LIN {X -0.034,Y -656.968,Z 952.580,A 0.000,B 0.000,C 90.000,E1 320.356} C_DIS
LIN {X 0.311,Y -657.904,Z 952.572,A 0.000,B 0.000,C 90.000,E1 318.852} C_DIS
LIN {X -0.424,Y -660.013,Z 952.555,A 0.000,B 0.000,C 90.000,E1 315.972} C_DIS
LIN {X -0.058,Y -660.986,Z 952.548,A 0.000,B 0.000,C 90.000,E1 314.717} C_DIS
LIN {X -0.144,Y -662.248,Z 952.540,A 0.000,B 0.000,C 90.000,E1 313.257} C_DIS
LIN {X 0.274,Y -663.376,Z 952.534,A 0.000,B 0.000,C 90.000,E1 312.000} C_DIS
LIN {X 0.265,Y -664.471,Z 952.527,A 0.000,B 0.000,C 90.000,E1 310.782} C_DIS
LIN {X 0.269,Y -665.467,Z 952.520,A 0.000,B 0.000,C 90.000,E1 309.564} C_DIS
LIN {X 0.361,Y -666.551,Z 952.512,A 0.000,B 0.000,C 90.000,E1 308.096} C_DIS
LIN {X 0.008,Y -666.996,Z 952.508,A 0.000,B 0.000,C 90.000,E1 307.397} C_DIS
LIN {X 0.120,Y -667.546,Z 952.500,A 0.000,B 0.000,C 90.000,E1 305.931} C_DIS
LIN {X -0.134,Y -667.856,Z 952.493,A 0.000,B 0.000,C 90.000,E1 304.739} C_DIS
LIN {X -0.167,Y -668.611,Z 952.482,A 0.000,B 0.000,C 90.000,E1 302.801} C_DIS
LIN {X 0.172,Y -669.793,Z 952.470,A 0.000,B 0.000,C 90.000,E1 300.590} C_DIS
LIN {X 0.063,Y -672.092,Z 952.457,A 0.000,B 0.000,C 90.000,E1 298.180} C_DIS
LIN {X 0.115,Y -676.639,Z 952.441,A 0.000,B 0.000,C 90.000,E1 295.283} C_DIS
LIN {X -0.028,Y -678.295,Z 952.435,A 0.000,B 0.000,C 90.000,E1 294.335} C_DIS
LIN {X -0.155,Y -679.852,Z 952.430,A 0.000,B 0.000,C 90.000,E1 293.387} C_DIS
LIN {X 0.161,Y -680.657,Z 952.426,A 0.000,B 0.000,C 90.000,E1 292.642} C_DIS
LIN {X 0.291,Y -680.615,Z 952.423,A 0.000,B 0.000,C 90.000,E1 292.153} C_DIS
LIN {X -0.147,Y -680.417,Z 952.422,A 0.000,B 0.000,C 90.000,E1 291.950} C_DIS
LIN {X -0.018,Y -679.161,Z 952.419,A 0.000,B 0.000,C 90.000,E1 291.461} C_DIS
LIN {X -0.078,Y -678.100,Z 952.418,A 0.000,B 0.000,C 90.000,E1 291.227} C_DIS
LIN {X 0.014,Y -677.207,Z 952.417,A 0.000,B 0.000,C 90.000,E1 291.099} C_DIS
LIN {X 0.256,Y -672.191,Z 952.415,A 0.000,B 0.000,C 90.000,E1 290.610} C_DIS
LIN {X 0.405,Y -670.668,Z 952.414,A 0.000,B 0.000,C 90.000,E1 290.482} C_DIS
LIN {X 0.041,Y -664.411,Z 952.412,A 0.000,B 0.000,C 90.000,E1 290.120} C_DIS
LIN {X -0.165,Y -660.787,Z 952.410,A 0.000,B 0.000,C 90.000,E1 289.885} C_DIS
LIN {X 0.054,Y -659.322,Z 952.410,A 0.000,B 0.000,C 90.000,E1 289.704} C_DIS
LIN {X 0.020,Y -659.313,Z 952.410,A 0.000,B 0.000,C 90.000,E1 289.704} C_DIS
LIN {X -0.271,Y -659.235,Z 952.409,A 0.000,B 0.000,C 90.000,E1 289.577} C_DIS
LIN {X 0.275,Y -660.197,Z 952.406,A 0.000,B 0.000,C 90.000,E1 289.141} C_DIS
LIN {X 0.110,Y -660.600,Z 952.406,A 0.000,B 0.000,C 90.000,E1 289.033} C_DIS
LIN {X 0.245,Y -663.941,Z 952.402,A 0.000,B 0.000,C 90.000,E1 288.362} C_DIS
LIN {X 0.096,Y -669.368,Z 952.397,A 0.000,B 0.000,C 90.000,E1 287.402} C_DIS
LIN {X 0.020,Y -670.659,Z 952.395,A 0.000,B 0.000,C 90.000,E1 287.166} C_DIS
LIN {X 0.010,Y -673.899,Z 952.391,A 0.000,B 0.000,C 90.000,E1 286.441} C_DIS
LIN {X -0.107,Y -675.770,Z 952.389,A 0.000,B 0.000,C 90.000,E1 285.969} C_DIS
LIN {X -0.079,Y -678.023,Z 952.385,A 0.000,B 0.000,C 90.000,E1 285.245} C_DIS
LIN {X -0.211,Y -679.726,Z 952.381,A 0.000,B 0.000,C 90.000,E1 284.537} C_DIS
LIN {X -0.324,Y -681.078,Z 952.377,A 0.000,B 0.000,C 90.000,E1 283.828} C_DIS
LIN {X 0.240,Y -682.253,Z 952.373,A 0.000,B 0.000,C 90.000,E1 283.063} C_DIS
LIN {X 0.149,Y -683.132,Z 952.369,A 0.000,B 0.000,C 90.000,E1 282.355} C_DIS
LIN {X -0.078,Y -683.629,Z 952.365,A 0.000,B 0.000,C 90.000,E1 281.658} C_DIS
LIN {X -0.134,Y -683.759,Z 952.362,A 0.000,B 0.000,C 90.000,E1 281.186} C_DIS
LIN {X -0.193,Y -683.585,Z 952.359,A 0.000,B 0.000,C 90.000,E1 280.715} C_DIS
LIN {X 0.293,Y -683.161,Z 952.357,A 0.000,B 0.000,C 90.000,E1 280.197} C_DIS
LIN {X 0.225,Y -682.382,Z 952.354,A 0.000,B 0.000,C 90.000,E1 279.726} C_DIS
LIN {X 0.038,Y -681.260,Z 952.352,A 0.000,B 0.000,C 90.000,E1 279.265} C_DIS
LIN {X -0.005,Y -680.643,Z 952.350,A 0.000,B 0.000,C 90.000,E1 279.029} C_DIS
LIN {X -0.200,Y -679.067,Z 952.348,A 0.000,B 0.000,C 90.000,E1 278.568} C_DIS
LIN {X 0.268,Y -677.154,Z 952.345,A 0.000,B 0.000,C 90.000,E1 278.049} C_DIS
LIN {X -0.011,Y -673.847,Z 952.341,A 0.000,B 0.000,C 90.000,E1 277.352} C_DIS
LIN {X -0.328,Y -670.649,Z 952.338,A 0.000,B 0.000,C 90.000,E1 276.777} C_DIS
LIN {X 0.083,Y -667.833,Z 952.335,A 0.000,B 0.000,C 90.000,E1 276.258} C_DIS
LIN {X -0.190,Y -664.711,Z 952.332,A 0.000,B 0.000,C 90.000,E1 275.796} C_DIS
LIN {X 0.175,Y -661.143,Z 952.329,A 0.000,B 0.000,C 90.000,E1 275.277} C_DIS
LIN {X -0.131,Y -657.252,Z 952.327,A 0.000,B 0.000,C 90.000,E1 274.821} C_DIS
LIN {X 0.082,Y -651.803,Z 952.323,A 0.000,B 0.000,C 90.000,E1 274.188} C_DIS
LIN {X 0.251,Y -645.769,Z 952.320,A 0.000,B 0.000,C 90.000,E1 273.555} C_DIS
LIN {X -0.042,Y -640.679,Z 952.317,A 0.000,B 0.000,C 90.000,E1 273.094} C_DIS
LIN {X -0.139,Y -634.030,Z 952.314,A 0.000,B 0.000,C 90.000,E1 272.522} C_DIS
LIN {X -0.082,Y -629.827,Z 952.312,A 0.000,B 0.000,C 90.000,E1 272.178} C_DIS
LIN {X 0.187,Y -623.963,Z 952.310,A 0.000,B 0.000,C 90.000,E1 271.718} C_DIS
LIN {X -0.114,Y -616.588,Z 952.307,A 0.000,B 0.000,C 90.000,E1 271.260} C_DIS
LIN {X 0.219,Y -610.478,Z 952.305,A 0.000,B 0.000,C 90.000,E1 270.859} C_DIS
LIN {X 0.009,Y -603.924,Z 952.303,A 0.000,B 0.000,C 90.000,E1 270.516} C_DIS
LIN {X 0.137,Y -597.098,Z 952.301,A 0.000,B 0.000,C 90.000,E1 270.172} C_DIS
LIN {X 0.154,Y -591.830,Z 952.300,A 0.000,B 0.000,C 90.000,E1 269.943} C_DIS
LIN {X -0.233,Y -584.711,Z 952.298,A 0.000,B 0.000,C 90.000,E1 269.714} C_DIS
LIN {X -0.222,Y -577.303,Z 952.297,A 0.000,B 0.000,C 90.000,E1 269.484} C_DIS
LIN {X 0.044,Y -571.553,Z 952.296,A 0.000,B 0.000,C 90.000,E1 269.312} C_DIS
LIN {X -0.073,Y -565.341,Z 952.296,A 0.000,B 0.000,C 90.000,E1 269.198} C_DIS
LIN {X 0.155,Y -558.224,Z 952.295,A 0.000,B 0.000,C 90.000,E1 269.083} C_DIS
LIN {X 0.117,Y -549.020,Z 952.295,A 0.000,B 0.000,C 90.000,E1 269.026} C_DIS
LIN {X 0.082,Y -548.656,Z 952.295,A 0.000,B 0.000,C 90.000,E1 269.026} C_DIS
LIN {X 0.048,Y -548.351,Z 952.295,A 0.000,B 0.000,C 90.000,E1 269.026} C_DIS
LIN {X 0.086,Y -545.265,Z 952.293,A 0.000,B 0.000,C 90.000,E1 268.797} C_DIS
LIN {X 0.116,Y -543.575,Z 952.293,A 0.000,B 0.000,C 90.000,E1 268.682} C_DIS
LIN {X 0.083,Y -543.532,Z 952.293,A 0.000,B 0.000,C 90.000,E1 268.682} C_DIS
LIN {X -0.111,Y -542.987,Z 952.291,A 0.000,B 0.000,C 90.000,E1 268.453} C_DIS
LIN {X -0.216,Y -541.694,Z 952.283,A 0.000,B 0.000,C 90.000,E1 266.906} C_DIS
LIN {X 0.018,Y -540.194,Z 952.272,A 0.000,B 0.000,C 90.000,E1 264.894} C_DIS
LIN {X 0.152,Y -539.180,Z 952.264,A 0.000,B 0.000,C 90.000,E1 263.457} C_DIS
LIN {X -0.140,Y -538.245,Z 952.256,A 0.000,B 0.000,C 90.000,E1 262.064} C_DIS
LIN {X 0.036,Y -537.214,Z 952.250,A 0.000,B 0.000,C 90.000,E1 260.905} C_DIS
LIN {X 0.132,Y -536.265,Z 952.245,A 0.000,B 0.000,C 90.000,E1 260.038} C_DIS
LIN {X -0.160,Y -534.759,Z 952.238,A 0.000,B 0.000,C 90.000,E1 258.926} C_DIS
LIN {X 0.150,Y -532.622,Z 952.229,A 0.000,B 0.000,C 90.000,E1 257.173} C_DIS
LIN {X 0.209,Y -529.843,Z 952.216,A 0.000,B 0.000,C 90.000,E1 254.866} C_DIS
LIN {X 0.141,Y -527.914,Z 952.206,A 0.000,B 0.000,C 90.000,E1 253.142} C_DIS
LIN {X 0.174,Y -525.866,Z 952.197,A 0.000,B 0.000,C 90.000,E1 251.402} C_DIS
LIN {X 0.173,Y -524.407,Z 952.190,A 0.000,B 0.000,C 90.000,E1 250.242} C_DIS
LIN {X 0.155,Y -522.900,Z 952.184,A 0.000,B 0.000,C 90.000,E1 249.082} C_DIS
LIN {X -0.068,Y -520.628,Z 952.174,A 0.000,B 0.000,C 90.000,E1 247.358} C_DIS
LIN {X 0.046,Y -518.967,Z 952.168,A 0.000,B 0.000,C 90.000,E1 246.177} C_DIS
LIN {X 0.142,Y -516.176,Z 952.158,A 0.000,B 0.000,C 90.000,E1 244.409} C_DIS
LIN {X 0.053,Y -513.862,Z 952.150,A 0.000,B 0.000,C 90.000,E1 242.948} C_DIS
LIN {X 0.042,Y -511.043,Z 952.140,A 0.000,B 0.000,C 90.000,E1 241.179} C_DIS
LIN {X 0.111,Y -509.554,Z 952.135,A 0.000,B 0.000,C 90.000,E1 240.284} C_DIS
LIN {X -0.182,Y -506.274,Z 952.125,A 0.000,B 0.000,C 90.000,E1 238.535} C_DIS
LIN {X -0.153,Y -503.051,Z 952.117,A 0.000,B 0.000,C 90.000,E1 237.041} C_DIS
LIN {X -0.082,Y -501.058,Z 952.112,A 0.000,B 0.000,C 90.000,E1 236.135} C_DIS
LIN {X 0.128,Y -497.613,Z 952.104,A 0.000,B 0.000,C 90.000,E1 234.609} C_DIS
LIN {X -0.280,Y -493.584,Z 952.093,A 0.000,B 0.000,C 90.000,E1 232.844} C_DIS
LIN {X -0.177,Y -489.479,Z 952.083,A 0.000,B 0.000,C 90.000,E1 231.009} C_DIS
LIN {X 0.173,Y -486.726,Z 952.077,A 0.000,B 0.000,C 90.000,E1 229.747} C_DIS
LIN {X -0.133,Y -481.730,Z 952.065,A 0.000,B 0.000,C 90.000,E1 227.634} C_DIS
LIN {X -0.077,Y -479.657,Z 952.059,A 0.000,B 0.000,C 90.000,E1 226.701} C_DIS
LIN {X -0.159,Y -476.262,Z 952.051,A 0.000,B 0.000,C 90.000,E1 225.162} C_DIS
LIN {X 0.317,Y -470.708,Z 952.037,A 0.000,B 0.000,C 90.000,E1 222.609} C_DIS
LIN {X 0.085,Y -467.334,Z 952.028,A 0.000,B 0.000,C 90.000,E1 221.067} C_DIS
LIN {X -0.065,Y -462.430,Z 952.016,A 0.000,B 0.000,C 90.000,E1 218.874} C_DIS
LIN {X -0.064,Y -459.673,Z 952.009,A 0.000,B 0.000,C 90.000,E1 217.604} C_DIS
LIN {X -0.088,Y -456.092,Z 952.000,A 0.000,B 0.000,C 90.000,E1 216.011} C_DIS
LIN {X -0.083,Y -452.498,Z 951.991,A 0.000,B 0.000,C 90.000,E1 214.405} C_DIS
LIN {X 0.226,Y -449.012,Z 951.982,A 0.000,B 0.000,C 90.000,E1 212.752} C_DIS
LIN {X -0.096,Y -444.823,Z 951.971,A 0.000,B 0.000,C 90.000,E1 210.846} C_DIS
LIN {X -0.110,Y -439.104,Z 951.957,A 0.000,B 0.000,C 90.000,E1 208.231} C_DIS
LIN {X 0.206,Y -436.270,Z 951.949,A 0.000,B 0.000,C 90.000,E1 206.873} C_DIS
LIN {X 0.102,Y -431.851,Z 951.938,A 0.000,B 0.000,C 90.000,E1 204.899} C_DIS
LIN {X -0.070,Y -428.864,Z 951.931,A 0.000,B 0.000,C 90.000,E1 203.590} C_DIS
LIN {X -0.122,Y -425.849,Z 951.924,A 0.000,B 0.000,C 90.000,E1 202.259} C_DIS
LIN {X -0.226,Y -419.995,Z 951.909,A 0.000,B 0.000,C 90.000,E1 199.577} C_DIS
LIN {X 0.153,Y -414.439,Z 951.893,A 0.000,B 0.000,C 90.000,E1 196.804} C_DIS
LIN {X -0.034,Y -410.348,Z 951.882,A 0.000,B 0.000,C 90.000,E1 194.773} C_DIS
LIN {X -0.142,Y -406.857,Z 951.872,A 0.000,B 0.000,C 90.000,E1 193.063} C_DIS
LIN {X 0.073,Y -403.492,Z 951.863,A 0.000,B 0.000,C 90.000,E1 191.299} C_DIS
LIN {X 0.060,Y -400.207,Z 951.853,A 0.000,B 0.000,C 90.000,E1 189.557} C_DIS
LIN {X -0.018,Y -396.831,Z 951.843,A 0.000,B 0.000,C 90.000,E1 187.814} C_DIS
LIN {X 0.085,Y -392.877,Z 951.832,A 0.000,B 0.000,C 90.000,E1 185.682} C_DIS
LIN {X 0.098,Y -387.044,Z 951.812,A 0.000,B 0.000,C 90.000,E1 182.121} C_DIS
LIN {X -0.084,Y -386.204,Z 951.808,A 0.000,B 0.000,C 90.000,E1 181.432} C_DIS
LIN {X 0.001,Y -385.558,Z 951.802,A 0.000,B 0.000,C 90.000,E1 180.344} C_DIS
LIN {X 0.182,Y -385.553,Z 951.798,A 0.000,B 0.000,C 90.000,E1 179.599} C_DIS
LIN {X 0.079,Y -385.809,Z 951.796,A 0.000,B 0.000,C 90.000,E1 179.255} C_DIS
LIN {X -0.076,Y -386.602,Z 951.793,A 0.000,B 0.000,C 90.000,E1 178.740} C_DIS
LIN {X 0.159,Y -387.894,Z 951.790,A 0.000,B 0.000,C 90.000,E1 178.167} C_DIS
LIN {X 0.119,Y -389.183,Z 951.788,A 0.000,B 0.000,C 90.000,E1 177.822} C_DIS
LIN {X 0.071,Y -390.016,Z 951.787,A 0.000,B 0.000,C 90.000,E1 177.650} C_DIS
LIN {X -0.106,Y -394.220,Z 951.783,A 0.000,B 0.000,C 90.000,E1 176.963} C_DIS
LIN {X -0.035,Y -400.464,Z 951.779,A 0.000,B 0.000,C 90.000,E1 176.274} C_DIS
LIN {X 0.135,Y -406.308,Z 951.776,A 0.000,B 0.000,C 90.000,E1 175.698} C_DIS
LIN {X 0.152,Y -413.777,Z 951.773,A 0.000,B 0.000,C 90.000,E1 175.065} C_DIS
LIN {X -0.174,Y -427.760,Z 951.766,A 0.000,B 0.000,C 90.000,E1 173.913} C_DIS
LIN {X -0.191,Y -436.865,Z 951.762,A 0.000,B 0.000,C 90.000,E1 173.109} C_DIS
LIN {X -0.015,Y -447.318,Z 951.756,A 0.000,B 0.000,C 90.000,E1 172.129} C_DIS
LIN {X 0.062,Y -457.365,Z 951.751,A 0.000,B 0.000,C 90.000,E1 171.141} C_DIS
LIN {X -0.080,Y -467.325,Z 951.745,A 0.000,B 0.000,C 90.000,E1 170.151} C_DIS
LIN {X -0.038,Y -469.990,Z 951.744,A 0.000,B 0.000,C 90.000,E1 169.859} C_DIS
LIN {X -0.150,Y -479.198,Z 951.738,A 0.000,B 0.000,C 90.000,E1 168.814} C_DIS
LIN {X -0.068,Y -485.493,Z 951.734,A 0.000,B 0.000,C 90.000,E1 168.049} C_DIS
LIN {X -0.135,Y -492.497,Z 951.729,A 0.000,B 0.000,C 90.000,E1 167.173} C_DIS
LIN {X 0.086,Y -501.659,Z 951.722,A 0.000,B 0.000,C 90.000,E1 165.936} C_DIS
LIN {X 0.070,Y -505.876,Z 951.719,A 0.000,B 0.000,C 90.000,E1 165.338} C_DIS
LIN {X 0.242,Y -510.876,Z 951.714,A 0.000,B 0.000,C 90.000,E1 164.574} C_DIS
LIN {X -0.036,Y -515.913,Z 951.710,A 0.000,B 0.000,C 90.000,E1 163.866} C_DIS
LIN {X 0.176,Y -523.464,Z 951.704,A 0.000,B 0.000,C 90.000,E1 162.670} C_DIS
LIN {X -0.167,Y -531.557,Z 951.697,A 0.000,B 0.000,C 90.000,E1 161.402} C_DIS
LIN {X -0.057,Y -538.744,Z 951.690,A 0.000,B 0.000,C 90.000,E1 160.242} C_DIS
LIN {X 0.063,Y -542.970,Z 951.686,A 0.000,B 0.000,C 90.000,E1 159.518} C_DIS
LIN {X 0.218,Y -550.595,Z 951.679,A 0.000,B 0.000,C 90.000,E1 158.230} C_DIS
LIN {X 0.306,Y -557.114,Z 951.673,A 0.000,B 0.000,C 90.000,E1 157.102} C_DIS
LIN {X -0.144,Y -562.448,Z 951.668,A 0.000,B 0.000,C 90.000,E1 156.177} C_DIS
LIN {X 0.020,Y -568.836,Z 951.661,A 0.000,B 0.000,C 90.000,E1 154.921} C_DIS
LIN {X 0.099,Y -572.209,Z 951.657,A 0.000,B 0.000,C 90.000,E1 154.229} C_DIS
LIN {X 0.154,Y -577.792,Z 951.650,A 0.000,B 0.000,C 90.000,E1 152.999} C_DIS
LIN {X -0.282,Y -581.356,Z 951.646,A 0.000,B 0.000,C 90.000,E1 152.231} C_DIS
LIN {X 0.099,Y -584.617,Z 951.641,A 0.000,B 0.000,C 90.000,E1 151.385} C_DIS
LIN {X -0.114,Y -588.762,Z 951.635,A 0.000,B 0.000,C 90.000,E1 150.333} C_DIS
LIN {X -0.079,Y -593.655,Z 951.628,A 0.000,B 0.000,C 90.000,E1 148.997} C_DIS
LIN {X 0.138,Y -597.398,Z 951.622,A 0.000,B 0.000,C 90.000,E1 147.916} C_DIS
LIN {X -0.184,Y -601.824,Z 951.615,A 0.000,B 0.000,C 90.000,E1 146.628} C_DIS
LIN {X -0.102,Y -606.319,Z 951.607,A 0.000,B 0.000,C 90.000,E1 145.308} C_DIS
LIN {X -0.232,Y -612.523,Z 951.597,A 0.000,B 0.000,C 90.000,E1 143.497} C_DIS
LIN {X 0.027,Y -618.611,Z 951.587,A 0.000,B 0.000,C 90.000,E1 141.662} C_DIS
LIN {X 0.266,Y -622.959,Z 951.580,A 0.000,B 0.000,C 90.000,E1 140.356} C_DIS
LIN {X 0.271,Y -632.602,Z 951.564,A 0.000,B 0.000,C 90.000,E1 137.553} C_DIS
LIN {X 0.199,Y -637.194,Z 951.557,A 0.000,B 0.000,C 90.000,E1 136.296} C_DIS
LIN {X -0.257,Y -641.762,Z 951.550,A 0.000,B 0.000,C 90.000,E1 135.081} C_DIS
LIN {X 0.273,Y -646.326,Z 951.543,A 0.000,B 0.000,C 90.000,E1 133.785} C_DIS
LIN {X -0.116,Y -652.727,Z 951.534,A 0.000,B 0.000,C 90.000,E1 132.081} C_DIS
LIN {X 0.135,Y -659.202,Z 951.524,A 0.000,B 0.000,C 90.000,E1 130.334} C_DIS
LIN {X 0.113,Y -665.712,Z 951.515,A 0.000,B 0.000,C 90.000,E1 128.624} C_DIS
LIN {X -0.283,Y -670.323,Z 951.508,A 0.000,B 0.000,C 90.000,E1 127.443} C_DIS
LIN {X -0.071,Y -673.781,Z 951.503,A 0.000,B 0.000,C 90.000,E1 126.457} C_DIS
LIN {X -0.356,Y -677.108,Z 951.497,A 0.000,B 0.000,C 90.000,E1 125.518} C_DIS
LIN {X 0.117,Y -680.941,Z 951.491,A 0.000,B 0.000,C 90.000,E1 124.278} C_DIS
LIN {X 0.088,Y -684.399,Z 951.484,A 0.000,B 0.000,C 90.000,E1 123.086} C_DIS
LIN {X 0.102,Y -686.975,Z 951.479,A 0.000,B 0.000,C 90.000,E1 122.133} C_DIS
LIN {X -0.211,Y -689.298,Z 951.473,A 0.000,B 0.000,C 90.000,E1 121.209} C_DIS
LIN {X 0.227,Y -690.889,Z 951.469,A 0.000,B 0.000,C 90.000,E1 120.463} C_DIS
LIN {X -0.271,Y -692.319,Z 951.465,A 0.000,B 0.000,C 90.000,E1 119.795} C_DIS
LIN {X 0.090,Y -693.838,Z 951.460,A 0.000,B 0.000,C 90.000,E1 118.821} C_DIS
LIN {X 0.224,Y -694.875,Z 951.456,A 0.000,B 0.000,C 90.000,E1 118.103} C_DIS
LIN {X 0.003,Y -695.819,Z 951.451,A 0.000,B 0.000,C 90.000,E1 117.180} C_DIS
LIN {X 0.351,Y -696.513,Z 951.445,A 0.000,B 0.000,C 90.000,E1 115.976} C_DIS
LIN {X 0.084,Y -696.830,Z 951.438,A 0.000,B 0.000,C 90.000,E1 114.823} C_DIS
LIN {X 0.309,Y -696.866,Z 951.435,A 0.000,B 0.000,C 90.000,E1 114.335} C_DIS
LIN {X -0.096,Y -696.657,Z 951.433,A 0.000,B 0.000,C 90.000,E1 113.898} C_DIS
LIN {X 0.161,Y -696.332,Z 951.431,A 0.000,B 0.000,C 90.000,E1 113.643} C_DIS
LIN {X -0.246,Y -695.305,Z 951.429,A 0.000,B 0.000,C 90.000,E1 113.206} C_DIS
LIN {X 0.005,Y -694.179,Z 951.428,A 0.000,B 0.000,C 90.000,E1 112.950} C_DIS
LIN {X 0.104,Y -692.115,Z 951.426,A 0.000,B 0.000,C 90.000,E1 112.589} C_DIS
LIN {X 0.224,Y -691.320,Z 951.425,A 0.000,B 0.000,C 90.000,E1 112.461} C_DIS
LIN {X 0.341,Y -690.170,Z 951.424,A 0.000,B 0.000,C 90.000,E1 112.333} C_DIS
LIN {X -0.179,Y -688.419,Z 951.424,A 0.000,B 0.000,C 90.000,E1 112.259} C_DIS
LIN {X -0.125,Y -681.797,Z 951.422,A 0.000,B 0.000,C 90.000,E1 111.897} C_DIS
LIN {X 0.030,Y -676.791,Z 951.421,A 0.000,B 0.000,C 90.000,E1 111.716} C_DIS
LIN {X 0.141,Y -674.368,Z 951.420,A 0.000,B 0.000,C 90.000,E1 111.663} C_DIS
LIN {X 0.298,Y -667.283,Z 951.420,A 0.000,B 0.000,C 90.000,E1 111.589} C_DIS
LIN {X 0.237,Y -633.015,Z 951.420,A 0.000,B 0.000,C 90.000,E1 111.589} C_DIS
LIN {X -0.285,Y -628.890,Z 951.420,A 0.000,B 0.000,C 90.000,E1 111.589} C_DIS
LIN {X 0.068,Y -623.504,Z 951.419,A 0.000,B 0.000,C 90.000,E1 111.461} C_DIS
LIN {X 0.141,Y -616.533,Z 951.418,A 0.000,B 0.000,C 90.000,E1 111.280} C_DIS
LIN {X 0.031,Y -612.934,Z 951.418,A 0.000,B 0.000,C 90.000,E1 111.173} C_DIS
LIN {X 0.242,Y -607.954,Z 951.417,A 0.000,B 0.000,C 90.000,E1 110.972} C_DIS
LIN {X -0.192,Y -599.704,Z 951.414,A 0.000,B 0.000,C 90.000,E1 110.610} C_DIS
LIN {X 0.171,Y -592.443,Z 951.412,A 0.000,B 0.000,C 90.000,E1 110.120} C_DIS
LIN {X 0.159,Y -576.614,Z 951.405,A 0.000,B 0.000,C 90.000,E1 108.960} C_DIS
LIN {X 0.143,Y -568.152,Z 951.403,A 0.000,B 0.000,C 90.000,E1 108.489} C_DIS
LIN {X 0.256,Y -557.668,Z 951.400,A 0.000,B 0.000,C 90.000,E1 108.000} C_DIS
LIN {X -0.160,Y -553.324,Z 951.399,A 0.000,B 0.000,C 90.000,E1 107.819} C_DIS
LIN {X -0.069,Y -551.566,Z 951.398,A 0.000,B 0.000,C 90.000,E1 107.638} C_DIS
LIN {X -0.102,Y -551.533,Z 951.398,A 0.000,B 0.000,C 90.000,E1 107.638} C_DIS
LIN {X -0.313,Y -551.046,Z 951.397,A 0.000,B 0.000,C 90.000,E1 107.402} C_DIS
LIN {X -0.082,Y -551.089,Z 951.393,A 0.000,B 0.000,C 90.000,E1 106.677} C_DIS
LIN {X 0.220,Y -551.640,Z 951.385,A 0.000,B 0.000,C 90.000,E1 105.245} C_DIS
LIN {X 0.085,Y -552.564,Z 951.374,A 0.000,B 0.000,C 90.000,E1 103.300} C_DIS
LIN {X 0.112,Y -554.362,Z 951.360,A 0.000,B 0.000,C 90.000,E1 100.782} C_DIS
LIN {X 0.203,Y -555.634,Z 951.352,A 0.000,B 0.000,C 90.000,E1 99.378} C_DIS
LIN {X 0.266,Y -557.104,Z 951.343,A 0.000,B 0.000,C 90.000,E1 97.701} C_DIS
LIN {X 0.229,Y -558.233,Z 951.335,A 0.000,B 0.000,C 90.000,E1 96.315} C_DIS
LIN {X -0.053,Y -558.817,Z 951.331,A 0.000,B 0.000,C 90.000,E1 95.511} C_DIS
LIN {X -0.197,Y -559.534,Z 951.324,A 0.000,B 0.000,C 90.000,E1 94.416} C_DIS
LIN {X -0.166,Y -560.482,Z 951.315,A 0.000,B 0.000,C 90.000,E1 92.751} C_DIS
LIN {X -0.241,Y -561.171,Z 951.308,A 0.000,B 0.000,C 90.000,E1 91.375} C_DIS
LIN {X 0.246,Y -561.730,Z 951.300,A 0.000,B 0.000,C 90.000,E1 89.943} C_DIS
LIN {X -0.018,Y -561.966,Z 951.295,A 0.000,B 0.000,C 90.000,E1 89.141} C_DIS
LIN {X 0.034,Y -562.318,Z 951.286,A 0.000,B 0.000,C 90.000,E1 87.478} C_DIS
LIN {X -0.203,Y -562.527,Z 951.281,A 0.000,B 0.000,C 90.000,E1 86.674} C_DIS
LIN {X -0.106,Y -562.806,Z 951.272,A 0.000,B 0.000,C 90.000,E1 85.008} C_DIS
LIN {X 0.129,Y -563.086,Z 951.262,A 0.000,B 0.000,C 90.000,E1 83.053} C_DIS
LIN {X -0.055,Y -563.492,Z 951.251,A 0.000,B 0.000,C 90.000,E1 81.141} C_DIS
LIN {X 0.205,Y -564.448,Z 951.237,A 0.000,B 0.000,C 90.000,E1 78.634} C_DIS
LIN {X -0.111,Y -565.643,Z 951.225,A 0.000,B 0.000,C 90.000,E1 76.464} C_DIS
LIN {X 0.103,Y -566.891,Z 951.214,A 0.000,B 0.000,C 90.000,E1 74.519} C_DIS
LIN {X 0.106,Y -568.138,Z 951.203,A 0.000,B 0.000,C 90.000,E1 72.598} C_DIS
LIN {X -0.018,Y -569.068,Z 951.194,A 0.000,B 0.000,C 90.000,E1 70.967} C_DIS
LIN {X -0.094,Y -569.586,Z 951.188,A 0.000,B 0.000,C 90.000,E1 69.880} C_DIS
LIN {X -0.009,Y -570.185,Z 951.179,A 0.000,B 0.000,C 90.000,E1 68.230} C_DIS
LIN {X -0.233,Y -570.641,Z 951.170,A 0.000,B 0.000,C 90.000,E1 66.613} C_DIS
LIN {X 0.134,Y -571.077,Z 951.159,A 0.000,B 0.000,C 90.000,E1 64.665} C_DIS
LIN {X 0.065,Y -571.303,Z 951.152,A 0.000,B 0.000,C 90.000,E1 63.307} C_DIS
LIN {X -0.259,Y -571.475,Z 951.144,A 0.000,B 0.000,C 90.000,E1 61.975} C_DIS
LIN {X -0.216,Y -571.498,Z 951.135,A 0.000,B 0.000,C 90.000,E1 60.333} C_DIS
LIN {X -0.057,Y -571.704,Z 951.125,A 0.000,B 0.000,C 90.000,E1 58.408} C_DIS
LIN {X -0.031,Y -571.588,Z 951.117,A 0.000,B 0.000,C 90.000,E1 57.041} C_DIS
LIN {X -0.008,Y -571.196,Z 951.109,A 0.000,B 0.000,C 90.000,E1 55.674} C_DIS
LIN {X 0.195,Y -570.844,Z 951.103,A 0.000,B 0.000,C 90.000,E1 54.562} C_DIS
LIN {X -0.204,Y -570.459,Z 951.099,A 0.000,B 0.000,C 90.000,E1 53.783} C_DIS
LIN {X 0.190,Y -569.991,Z 951.094,A 0.000,B 0.000,C 90.000,E1 52.924} C_DIS
LIN {X 0.257,Y -569.100,Z 951.088,A 0.000,B 0.000,C 90.000,E1 51.823} C_DIS
LIN {X 0.314,Y -568.029,Z 951.082,A 0.000,B 0.000,C 90.000,E1 50.723} C_DIS
LIN {X -0.080,Y -566.755,Z 951.076,A 0.000,B 0.000,C 90.000,E1 49.666} C_DIS
LIN {X -0.173,Y -565.633,Z 951.071,A 0.000,B 0.000,C 90.000,E1 48.852} C_DIS
LIN {X -0.009,Y -564.773,Z 951.068,A 0.000,B 0.000,C 90.000,E1 48.286} C_DIS
LIN {X 0.024,Y -562.164,Z 951.061,A 0.000,B 0.000,C 90.000,E1 46.905} C_DIS
LIN {X 0.249,Y -560.362,Z 951.056,A 0.000,B 0.000,C 90.000,E1 46.053} C_DIS
LIN {X 0.052,Y -558.253,Z 951.051,A 0.000,B 0.000,C 90.000,E1 45.243} C_DIS
LIN {X -0.166,Y -555.878,Z 951.047,A 0.000,B 0.000,C 90.000,E1 44.433} C_DIS
LIN {X -0.008,Y -553.216,Z 951.042,A 0.000,B 0.000,C 90.000,E1 43.581} C_DIS
LIN {X 0.075,Y -551.307,Z 951.039,A 0.000,B 0.000,C 90.000,E1 43.014} C_DIS
LIN {X 0.140,Y -549.224,Z 951.036,A 0.000,B 0.000,C 90.000,E1 42.447} C_DIS
LIN {X -0.179,Y -546.986,Z 951.033,A 0.000,B 0.000,C 90.000,E1 41.919} C_DIS
LIN {X -0.313,Y -543.886,Z 951.029,A 0.000,B 0.000,C 90.000,E1 41.229} C_DIS
LIN {X 0.285,Y -540.457,Z 951.025,A 0.000,B 0.000,C 90.000,E1 40.458} C_DIS
LIN {X 0.081,Y -536.745,Z 951.021,A 0.000,B 0.000,C 90.000,E1 39.769} C_DIS
LIN {X -0.079,Y -532.770,Z 951.017,A 0.000,B 0.000,C 90.000,E1 39.072} C_DIS
LIN {X 0.066,Y -528.586,Z 951.013,A 0.000,B 0.000,C 90.000,E1 38.338} C_DIS
LIN {X 0.137,Y -522.424,Z 951.007,A 0.000,B 0.000,C 90.000,E1 37.317} C_DIS
LIN {X 0.178,Y -517.744,Z 951.003,A 0.000,B 0.000,C 90.000,E1 36.583} C_DIS
LIN {X -0.016,Y -511.775,Z 950.999,A 0.000,B 0.000,C 90.000,E1 35.724} C_DIS
LIN {X 0.234,Y -507.552,Z 950.995,A 0.000,B 0.000,C 90.000,E1 35.105} C_DIS
LIN {X -0.158,Y -501.920,Z 950.991,A 0.000,B 0.000,C 90.000,E1 34.405} C_DIS
LIN {X 0.018,Y -496.996,Z 950.988,A 0.000,B 0.000,C 90.000,E1 33.785} C_DIS
LIN {X 0.041,Y -490.414,Z 950.984,A 0.000,B 0.000,C 90.000,E1 33.038} C_DIS
LIN {X -0.239,Y -486.249,Z 950.981,A 0.000,B 0.000,C 90.000,E1 32.625} C_DIS
LIN {X 0.105,Y -479.220,Z 950.977,A 0.000,B 0.000,C 90.000,E1 31.878} C_DIS
LIN {X -0.035,Y -473.456,Z 950.974,A 0.000,B 0.000,C 90.000,E1 31.337} C_DIS
LIN {X -0.014,Y -463.061,Z 950.969,A 0.000,B 0.000,C 90.000,E1 30.384} C_DIS
LIN {X -0.014,Y -455.532,Z 950.965,A 0.000,B 0.000,C 90.000,E1 29.716} C_DIS
LIN {X -0.147,Y -444.849,Z 950.960,A 0.000,B 0.000,C 90.000,E1 28.821} C_DIS
LIN {X 0.123,Y -424.991,Z 950.951,A 0.000,B 0.000,C 90.000,E1 27.078} C_DIS
LIN {X -0.014,Y -410.316,Z 950.943,A 0.000,B 0.000,C 90.000,E1 25.720} C_DIS
LIN {X -0.118,Y -400.108,Z 950.937,A 0.000,B 0.000,C 90.000,E1 24.695} C_DIS
LIN {X 0.184,Y -397.292,Z 950.935,A 0.000,B 0.000,C 90.000,E1 24.335} C_DIS
LIN {X 0.124,Y -393.895,Z 950.933,A 0.000,B 0.000,C 90.000,E1 23.898} C_DIS
LIN {X -0.121,Y -391.584,Z 950.931,A 0.000,B 0.000,C 90.000,E1 23.515} C_DIS
LIN {X -0.099,Y -390.911,Z 950.930,A 0.000,B 0.000,C 90.000,E1 23.334} C_DIS
LIN {X 0.096,Y -389.941,Z 950.928,A 0.000,B 0.000,C 90.000,E1 22.950} C_DIS
LIN {X -0.211,Y -389.319,Z 950.925,A 0.000,B 0.000,C 90.000,E1 22.461} C_DIS
LIN {X -0.029,Y -389.257,Z 950.923,A 0.000,B 0.000,C 90.000,E1 22.078} C_DIS
LIN {X 0.039,Y -389.556,Z 950.919,A 0.000,B 0.000,C 90.000,E1 21.354} C_DIS
LIN {X -0.034,Y -394.270,Z 950.891,A 0.000,B 0.000,C 90.000,E1 16.386} C_DIS
LIN {X 0.142,Y -397.820,Z 950.875,A 0.000,B 0.000,C 90.000,E1 13.536} C_DIS
LIN {X -0.166,Y -402.473,Z 950.858,A 0.000,B 0.000,C 90.000,E1 10.423} C_DIS
LIN {X 0.178,Y -406.596,Z 950.844,A 0.000,B 0.000,C 90.000,E1 7.936} C_DIS
LIN {X -0.206,Y -411.070,Z 950.831,A 0.000,B 0.000,C 90.000,E1 5.568} C_DIS
LIN {X -0.101,Y -416.770,Z 950.816,A 0.000,B 0.000,C 90.000,E1 2.808} C_DIS
LIN {X 0.208,Y -424.699,Z 950.797,A 0.000,B 0.000,C 90.000,E1 359.427} C_DIS
LIN {X -0.169,Y -425.664,Z 950.795,A 0.000,B 0.000,C 90.000,E1 359.141} C_DIS
LIN {X -0.058,Y -428.568,Z 950.791,A 0.000,B 0.000,C 90.000,E1 358.453} C_DIS
LIN {X 0.204,Y -430.928,Z 950.789,A 0.000,B 0.000,C 90.000,E1 358.051} C_DIS
LIN {X -0.194,Y -432.326,Z 950.788,A 0.000,B 0.000,C 90.000,E1 357.936} C_DIS
LIN {X 0.095,Y -435.439,Z 950.787,A 0.000,B 0.000,C 90.000,E1 357.593} C_DIS
LIN {X -0.080,Y -441.046,Z 950.785,A 0.000,B 0.000,C 90.000,E1 357.249} C_DIS
LIN {X -0.097,Y -459.223,Z 950.780,A 0.000,B 0.000,C 90.000,E1 356.331} C_DIS
LIN {X 0.093,Y -467.451,Z 950.777,A 0.000,B 0.000,C 90.000,E1 355.869} C_DIS
LIN {X -0.116,Y -477.712,Z 950.774,A 0.000,B 0.000,C 90.000,E1 355.355} C_DIS
LIN {X -0.230,Y -490.664,Z 950.770,A 0.000,B 0.000,C 90.000,E1 354.666} C_DIS
LIN {X 0.097,Y -497.376,Z 950.768,A 0.000,B 0.000,C 90.000,E1 354.261} C_DIS
LIN {X -0.128,Y -508.610,Z 950.765,A 0.000,B 0.000,C 90.000,E1 353.628} C_DIS
LIN {X 0.139,Y -518.302,Z 950.761,A 0.000,B 0.000,C 90.000,E1 352.996} C_DIS
LIN {X 0.245,Y -527.485,Z 950.758,A 0.000,B 0.000,C 90.000,E1 352.356} C_DIS
LIN {X -0.128,Y -534.883,Z 950.755,A 0.000,B 0.000,C 90.000,E1 351.837} C_DIS
LIN {X -0.151,Y -542.063,Z 950.751,A 0.000,B 0.000,C 90.000,E1 351.254} C_DIS
LIN {X -0.041,Y -548.884,Z 950.748,A 0.000,B 0.000,C 90.000,E1 350.622} C_DIS
LIN {X -0.253,Y -555.249,Z 950.744,A 0.000,B 0.000,C 90.000,E1 349.982} C_DIS
LIN {X -0.204,Y -559.032,Z 950.742,A 0.000,B 0.000,C 90.000,E1 349.567} C_DIS
LIN {X -0.120,Y -564.741,Z 950.738,A 0.000,B 0.000,C 90.000,E1 348.870} C_DIS
LIN {X -0.033,Y -570.014,Z 950.734,A 0.000,B 0.000,C 90.000,E1 348.173} C_DIS
LIN {X -0.220,Y -573.957,Z 950.731,A 0.000,B 0.000,C 90.000,E1 347.645} C_DIS
LIN {X -0.170,Y -579.426,Z 950.727,A 0.000,B 0.000,C 90.000,E1 346.825} C_DIS
LIN {X 0.173,Y -583.556,Z 950.723,A 0.000,B 0.000,C 90.000,E1 346.117} C_DIS
LIN {X 0.149,Y -589.826,Z 950.717,A 0.000,B 0.000,C 90.000,E1 345.046} C_DIS
LIN {X -0.287,Y -594.799,Z 950.712,A 0.000,B 0.000,C 90.000,E1 344.157} C_DIS
LIN {X -0.159,Y -600.112,Z 950.706,A 0.000,B 0.000,C 90.000,E1 343.087} C_DIS
LIN {X -0.309,Y -604.499,Z 950.701,A 0.000,B 0.000,C 90.000,E1 342.181} C_DIS
LIN {X 0.167,Y -608.706,Z 950.696,A 0.000,B 0.000,C 90.000,E1 341.221} C_DIS
LIN {X 0.345,Y -612.125,Z 950.691,A 0.000,B 0.000,C 90.000,E1 340.423} C_DIS
LIN {X 0.057,Y -617.430,Z 950.684,A 0.000,B 0.000,C 90.000,E1 339.156} C_DIS
LIN {X -0.250,Y -620.426,Z 950.680,A 0.000,B 0.000,C 90.000,E1 338.411} C_DIS
LIN {X 0.045,Y -625.117,Z 950.673,A 0.000,B 0.000,C 90.000,E1 337.102} C_DIS
LIN {X -0.148,Y -629.444,Z 950.666,A 0.000,B 0.000,C 90.000,E1 335.845} C_DIS
LIN {X 0.301,Y -633.403,Z 950.659,A 0.000,B 0.000,C 90.000,E1 334.537} C_DIS
LIN {X -0.056,Y -637.032,Z 950.652,A 0.000,B 0.000,C 90.000,E1 333.307} C_DIS
LIN {X 0.160,Y -639.735,Z 950.646,A 0.000,B 0.000,C 90.000,E1 332.281} C_DIS
LIN {X -0.157,Y -642.155,Z 950.641,A 0.000,B 0.000,C 90.000,E1 331.307} C_DIS
LIN {X -0.058,Y -645.026,Z 950.634,A 0.000,B 0.000,C 90.000,E1 330.049} C_DIS
LIN {X 0.091,Y -647.561,Z 950.627,A 0.000,B 0.000,C 90.000,E1 328.791} C_DIS
LIN {X -0.279,Y -649.695,Z 950.620,A 0.000,B 0.000,C 90.000,E1 327.582} C_DIS
LIN {X -0.161,Y -651.256,Z 950.614,A 0.000,B 0.000,C 90.000,E1 326.580} C_DIS
LIN {X 0.239,Y -652.864,Z 950.607,A 0.000,B 0.000,C 90.000,E1 325.308} C_DIS
LIN {X -0.230,Y -653.793,Z 950.603,A 0.000,B 0.000,C 90.000,E1 324.609} C_DIS
LIN {X 0.222,Y -654.934,Z 950.596,A 0.000,B 0.000,C 90.000,E1 323.336} C_DIS
LIN {X 0.167,Y -655.981,Z 950.590,A 0.000,B 0.000,C 90.000,E1 322.110} C_DIS
LIN {X -0.383,Y -657.267,Z 950.580,A 0.000,B 0.000,C 90.000,E1 320.436} C_DIS
LIN {X -0.034,Y -658.233,Z 950.572,A 0.000,B 0.000,C 90.000,E1 318.933} C_DIS
LIN {X 0.174,Y -660.354,Z 950.556,A 0.000,B 0.000,C 90.000,E1 315.972} C_DIS
LIN {X 0.082,Y -661.334,Z 950.549,A 0.000,B 0.000,C 90.000,E1 314.757} C_DIS
LIN {X -0.044,Y -663.079,Z 950.538,A 0.000,B 0.000,C 90.000,E1 312.813} C_DIS
LIN {X 0.401,Y -664.625,Z 950.528,A 0.000,B 0.000,C 90.000,E1 311.067} C_DIS
LIN {X -0.035,Y -665.855,Z 950.520,A 0.000,B 0.000,C 90.000,E1 309.644} C_DIS
LIN {X 0.066,Y -666.970,Z 950.512,A 0.000,B 0.000,C 90.000,E1 308.177} C_DIS
LIN {X 0.124,Y -667.448,Z 950.508,A 0.000,B 0.000,C 90.000,E1 307.443} C_DIS
LIN {X 0.267,Y -667.930,Z 950.501,A 0.000,B 0.000,C 90.000,E1 306.217} C_DIS
LIN {X 0.149,Y -668.336,Z 950.493,A 0.000,B 0.000,C 90.000,E1 304.771} C_DIS
LIN {X 0.149,Y -669.081,Z 950.483,A 0.000,B 0.000,C 90.000,E1 302.832} C_DIS
LIN {X 0.207,Y -669.940,Z 950.473,A 0.000,B 0.000,C 90.000,E1 301.131} C_DIS
LIN {X 0.107,Y -673.479,Z 950.453,A 0.000,B 0.000,C 90.000,E1 297.513} C_DIS
LIN {X 0.233,Y -677.027,Z 950.441,A 0.000,B 0.000,C 90.000,E1 295.335} C_DIS
LIN {X 0.004,Y -679.068,Z 950.434,A 0.000,B 0.000,C 90.000,E1 294.155} C_DIS
LIN {X -0.036,Y -680.215,Z 950.430,A 0.000,B 0.000,C 90.000,E1 293.439} C_DIS
LIN {X 0.018,Y -681.028,Z 950.426,A 0.000,B 0.000,C 90.000,E1 292.717} C_DIS
LIN {X 0.410,Y -681.017,Z 950.424,A 0.000,B 0.000,C 90.000,E1 292.206} C_DIS
LIN {X -0.281,Y -680.920,Z 950.422,A 0.000,B 0.000,C 90.000,E1 292.025} C_DIS
LIN {X -0.088,Y -680.377,Z 950.421,A 0.000,B 0.000,C 90.000,E1 291.770} C_DIS
LIN {X -0.146,Y -679.618,Z 950.420,A 0.000,B 0.000,C 90.000,E1 291.535} C_DIS
LIN {X 0.044,Y -678.547,Z 950.418,A 0.000,B 0.000,C 90.000,E1 291.280} C_DIS
LIN {X 0.135,Y -677.834,Z 950.418,A 0.000,B 0.000,C 90.000,E1 291.153} C_DIS
LIN {X -0.015,Y -676.771,Z 950.417,A 0.000,B 0.000,C 90.000,E1 291.046} C_DIS
LIN {X 0.314,Y -672.851,Z 950.415,A 0.000,B 0.000,C 90.000,E1 290.663} C_DIS
LIN {X 0.230,Y -671.412,Z 950.414,A 0.000,B 0.000,C 90.000,E1 290.556} C_DIS
LIN {X 0.200,Y -663.724,Z 950.412,A 0.000,B 0.000,C 90.000,E1 290.066} C_DIS
LIN {X 0.068,Y -660.985,Z 950.411,A 0.000,B 0.000,C 90.000,E1 289.885} C_DIS
LIN {X 0.027,Y -659.732,Z 950.410,A 0.000,B 0.000,C 90.000,E1 289.758} C_DIS
LIN {X -0.010,Y -659.719,Z 950.410,A 0.000,B 0.000,C 90.000,E1 289.758} C_DIS
LIN {X -0.093,Y -659.783,Z 950.409,A 0.000,B 0.000,C 90.000,E1 289.577} C_DIS
LIN {X -0.040,Y -659.945,Z 950.408,A 0.000,B 0.000,C 90.000,E1 289.450} C_DIS
LIN {X -0.338,Y -661.118,Z 950.406,A 0.000,B 0.000,C 90.000,E1 289.087} C_DIS
LIN {X 0.194,Y -664.890,Z 950.402,A 0.000,B 0.000,C 90.000,E1 288.308} C_DIS
LIN {X 0.199,Y -669.570,Z 950.397,A 0.000,B 0.000,C 90.000,E1 287.457} C_DIS
LIN {X 0.185,Y -671.452,Z 950.395,A 0.000,B 0.000,C 90.000,E1 287.094} C_DIS
LIN {X -0.013,Y -674.609,Z 950.391,A 0.000,B 0.000,C 90.000,E1 286.386} C_DIS
LIN {X 0.061,Y -676.420,Z 950.388,A 0.000,B 0.000,C 90.000,E1 285.898} C_DIS
LIN {X -0.087,Y -678.586,Z 950.384,A 0.000,B 0.000,C 90.000,E1 285.190} C_DIS
LIN {X -0.172,Y -679.772,Z 950.382,A 0.000,B 0.000,C 90.000,E1 284.717} C_DIS
LIN {X -0.283,Y -681.196,Z 950.378,A 0.000,B 0.000,C 90.000,E1 284.008} C_DIS
LIN {X 0.283,Y -682.407,Z 950.374,A 0.000,B 0.000,C 90.000,E1 283.244} C_DIS
LIN {X 0.198,Y -683.369,Z 950.370,A 0.000,B 0.000,C 90.000,E1 282.535} C_DIS
LIN {X 0.116,Y -684.052,Z 950.366,A 0.000,B 0.000,C 90.000,E1 281.827} C_DIS
LIN {X -0.076,Y -684.273,Z 950.363,A 0.000,B 0.000,C 90.000,E1 281.366} C_DIS
LIN {X -0.156,Y -684.097,Z 950.359,A 0.000,B 0.000,C 90.000,E1 280.658} C_DIS
LIN {X -0.338,Y -683.677,Z 950.357,A 0.000,B 0.000,C 90.000,E1 280.197} C_DIS
LIN {X 0.271,Y -682.820,Z 950.354,A 0.000,B 0.000,C 90.000,E1 279.670} C_DIS
LIN {X 0.087,Y -681.669,Z 950.351,A 0.000,B 0.000,C 90.000,E1 279.208} C_DIS
LIN {X 0.046,Y -681.019,Z 950.350,A 0.000,B 0.000,C 90.000,E1 278.973} C_DIS
LIN {X -0.146,Y -679.405,Z 950.347,A 0.000,B 0.000,C 90.000,E1 278.511} C_DIS
LIN {X -0.346,Y -677.407,Z 950.345,A 0.000,B 0.000,C 90.000,E1 278.049} C_DIS
LIN {X 0.049,Y -674.001,Z 950.341,A 0.000,B 0.000,C 90.000,E1 277.296} C_DIS
LIN {X -0.182,Y -671.506,Z 950.338,A 0.000,B 0.000,C 90.000,E1 276.834} C_DIS
LIN {X 0.148,Y -667.981,Z 950.335,A 0.000,B 0.000,C 90.000,E1 276.201} C_DIS
LIN {X -0.036,Y -665.719,Z 950.333,A 0.000,B 0.000,C 90.000,E1 275.853} C_DIS
LIN {X 0.243,Y -661.253,Z 950.329,A 0.000,B 0.000,C 90.000,E1 275.220} C_DIS
LIN {X -0.075,Y -657.366,Z 950.326,A 0.000,B 0.000,C 90.000,E1 274.759} C_DIS
LIN {X 0.170,Y -651.899,Z 950.323,A 0.000,B 0.000,C 90.000,E1 274.131} C_DIS
LIN {X -0.206,Y -647.154,Z 950.320,A 0.000,B 0.000,C 90.000,E1 273.669} C_DIS
LIN {X 0.095,Y -642.163,Z 950.318,A 0.000,B 0.000,C 90.000,E1 273.154} C_DIS
LIN {X -0.056,Y -635.498,Z 950.314,A 0.000,B 0.000,C 90.000,E1 272.579} C_DIS
LIN {X -0.010,Y -631.424,Z 950.312,A 0.000,B 0.000,C 90.000,E1 272.236} C_DIS
LIN {X 0.291,Y -624.034,Z 950.309,A 0.000,B 0.000,C 90.000,E1 271.661} C_DIS
LIN {X 0.027,Y -616.662,Z 950.307,A 0.000,B 0.000,C 90.000,E1 271.203} C_DIS
LIN {X 0.250,Y -610.418,Z 950.305,A 0.000,B 0.000,C 90.000,E1 270.802} C_DIS
LIN {X 0.094,Y -603.885,Z 950.303,A 0.000,B 0.000,C 90.000,E1 270.458} C_DIS
LIN {X 0.218,Y -597.077,Z 950.301,A 0.000,B 0.000,C 90.000,E1 270.115} C_DIS
LIN {X 0.244,Y -591.808,Z 950.300,A 0.000,B 0.000,C 90.000,E1 269.885} C_DIS
LIN {X -0.166,Y -584.689,Z 950.298,A 0.000,B 0.000,C 90.000,E1 269.656} C_DIS
LIN {X -0.176,Y -577.044,Z 950.297,A 0.000,B 0.000,C 90.000,E1 269.427} C_DIS
LIN {X 0.111,Y -571.272,Z 950.296,A 0.000,B 0.000,C 90.000,E1 269.255} C_DIS
LIN {X 0.013,Y -565.113,Z 950.295,A 0.000,B 0.000,C 90.000,E1 269.141} C_DIS
LIN {X 0.263,Y -557.874,Z 950.295,A 0.000,B 0.000,C 90.000,E1 269.026} C_DIS
LIN {X -0.182,Y -550.210,Z 950.295,A 0.000,B 0.000,C 90.000,E1 269.026} C_DIS
LIN {X 0.185,Y -548.531,Z 950.294,A 0.000,B 0.000,C 90.000,E1 268.969} C_DIS
LIN {X 0.149,Y -548.311,Z 950.294,A 0.000,B 0.000,C 90.000,E1 268.969} C_DIS
LIN {X 0.093,Y -546.585,Z 950.294,A 0.000,B 0.000,C 90.000,E1 268.854} C_DIS
LIN {X 0.151,Y -543.780,Z 950.293,A 0.000,B 0.000,C 90.000,E1 268.682} C_DIS
LIN {X 0.095,Y -543.712,Z 950.293,A 0.000,B 0.000,C 90.000,E1 268.682} C_DIS
LIN {X 0.245,Y -543.075,Z 950.291,A 0.000,B 0.000,C 90.000,E1 268.396} C_DIS
LIN {X 0.140,Y -541.772,Z 950.283,A 0.000,B 0.000,C 90.000,E1 266.849} C_DIS
LIN {X -0.165,Y -540.273,Z 950.272,A 0.000,B 0.000,C 90.000,E1 264.894} C_DIS
LIN {X 0.032,Y -539.259,Z 950.264,A 0.000,B 0.000,C 90.000,E1 263.451} C_DIS
LIN {X 0.215,Y -538.311,Z 950.256,A 0.000,B 0.000,C 90.000,E1 262.008} C_DIS
LIN {X -0.142,Y -537.317,Z 950.249,A 0.000,B 0.000,C 90.000,E1 260.905} C_DIS
LIN {X -0.044,Y -536.355,Z 950.245,A 0.000,B 0.000,C 90.000,E1 260.038} C_DIS
LIN {X 0.191,Y -534.834,Z 950.238,A 0.000,B 0.000,C 90.000,E1 258.870} C_DIS
LIN {X -0.021,Y -532.661,Z 950.229,A 0.000,B 0.000,C 90.000,E1 257.173} C_DIS
LIN {X 0.039,Y -529.905,Z 950.216,A 0.000,B 0.000,C 90.000,E1 254.866} C_DIS
LIN {X -0.027,Y -527.962,Z 950.206,A 0.000,B 0.000,C 90.000,E1 253.142} C_DIS
LIN {X 0.005,Y -526.254,Z 950.198,A 0.000,B 0.000,C 90.000,E1 251.692} C_DIS
LIN {X -0.158,Y -524.805,Z 950.192,A 0.000,B 0.000,C 90.000,E1 250.550} C_DIS
LIN {X -0.010,Y -522.922,Z 950.184,A 0.000,B 0.000,C 90.000,E1 249.082} C_DIS
END
